(* PLC project emC-LUC-BS-Temp, PHOENIX CONTACT Software MULTIPROG 5.51 *)
(* stored: companyURL https://www.phoenixcontact-software.com, creationDateTime 2020-12-01T16:35:25, version 1606836925, modificationDateTime 2020-12-01T16:35:25 *)

TYPE TDC_DATA : ARRAY[0..199] OF BYTE;
END_TYPE

TYPE TDC : STRUCT
  transmit : BOOL;
  COT : USINT;
  confirm : BOOL;
  COTDesc : USINT;
  intOriginator : USINT;
  protocolType : USINT;
  totalNoOfSegments : USINT;
  currentSegment : USINT;
  lenOfData : UINT;
  data : TDC_DATA;
END_STRUCT;
END_TYPE

TYPE ThresholdType : (None, Integrated, Absolute) INT;
END_TYPE

TYPE COT : STRUCT
  Act : BOOL;
  ActCon : BOOL;
  Deact : BOOL;
  DeactCon : BOOL;
  ActTerm : BOOL;
END_STRUCT;
END_TYPE

TYPE Timestamp : STRUCT
  Milliseconds : UINT;
  Minutes : USINT;
  IV : BOOL;
  Hours : USINT;
  Summertime : BOOL;
  DayOfMonth : USINT;
  DayOfWeek : USINT;
  Month : USINT;
  Year : USINT;
END_STRUCT;
END_TYPE

TYPE AMI : STRUCT
  Value : INT;
  OV : BOOL;
  BL : BOOL;
  SB : BOOL;
  NT : BOOL;
  IV : BOOL;
  TR : BOOL;
  TimeTag : Timestamp;
  COT : USINT;
  FILL : BOOL;
END_STRUCT;
END_TYPE

TYPE ASO : STRUCT
  SE : BOOL;
  EX : BOOL;
  AQ : BOOL;
  QU : BYTE;
  Value : INT;
  COT : USINT;
  COTDesc : USINT;
  intOriginator : USINT;
END_STRUCT;
END_TYPE

TYPE BSI08 : STRUCT
  Value : BYTE;
  OV : BOOL;
  BL : BOOL;
  SB : BOOL;
  NT : BOOL;
  IV : BOOL;
  TimeTag : Timestamp;
  COT : USINT;
  FILL : BOOL;
END_STRUCT;
END_TYPE

TYPE BSI16 : STRUCT
  Value : WORD;
  OV : BOOL;
  BL : BOOL;
  SB : BOOL;
  NT : BOOL;
  IV : BOOL;
  FILL1 : BOOL;
  TimeTag : Timestamp;
  COT : USINT;
  FILL2 : BOOL;
END_STRUCT;
END_TYPE

TYPE BSI32 : STRUCT
  Value : DWORD;
  OV : BOOL;
  BL : BOOL;
  SB : BOOL;
  NT : BOOL;
  IV : BOOL;
  FILL1 : BOOL;
  TimeTag : Timestamp;
  COT : USINT;
  FILL2 : BOOL;
END_STRUCT;
END_TYPE

TYPE BSO01 : STRUCT
  SE : BOOL;
  EX : BOOL;
  AQ : BOOL;
  QU : BYTE;
  Value : BOOL;
  COT : USINT;
  COTDesc : USINT;
  intOriginator : USINT;
END_STRUCT;
END_TYPE

TYPE BSO02 : STRUCT
  SE : BOOL;
  EX : BOOL;
  AQ : BOOL;
  QU : BYTE;
  Value : BYTE;
  COT : USINT;
  COTDesc : USINT;
  intOriginator : USINT;
END_STRUCT;
END_TYPE

TYPE BSO08 : STRUCT
  SE : BOOL;
  EX : BOOL;
  AQ : BOOL;
  QU : BYTE;
  Value : BYTE;
  COT : USINT;
  COTDesc : USINT;
  intOriginator : USINT;
END_STRUCT;
END_TYPE

TYPE BSO16 : STRUCT
  SE : BOOL;
  EX : BOOL;
  AQ : BOOL;
  QU : BYTE;
  Value : WORD;
  COT : USINT;
  COTDesc : USINT;
  intOriginator : USINT;
END_STRUCT;
END_TYPE

TYPE DCO : STRUCT
  SE : BOOL;
  EX : BOOL;
  AQ : BOOL;
  QU : BYTE;
  Value : BYTE;
  COT : USINT;
  COTDesc : USINT;
  intOriginator : USINT;
END_STRUCT;
END_TYPE

TYPE DMI08 : STRUCT
  Value : WORD;
  OV : BOOL;
  BL : BOOL;
  SB : BOOL;
  NT : BOOL;
  IV : BOOL;
  FILL1 : BOOL;
  TimeTag : Timestamp;
  COT : USINT;
  FILL2 : BOOL;
END_STRUCT;
END_TYPE

TYPE DMI16 : STRUCT
  Value : WORD;
  OV : BOOL;
  BL : BOOL;
  SB : BOOL;
  NT : BOOL;
  IV : BOOL;
  FILL1 : BOOL;
  TimeTag : Timestamp;
  COT : USINT;
  FILL2 : BOOL;
END_STRUCT;
END_TYPE

TYPE DPI : STRUCT
  Value : BYTE;
  BL : BOOL;
  SB : BOOL;
  NT : BOOL;
  IV : BOOL;
  FILL1 : BOOL;
  TimeTag : Timestamp;
  COT : USINT;
  FILL2 : BOOL;
END_STRUCT;
END_TYPE

TYPE DSO08 : STRUCT
  SE : BOOL;
  EX : BOOL;
  AQ : BOOL;
  QU : BYTE;
  Value : INT;
  COT : USINT;
  COTDesc : USINT;
  intOriginator : USINT;
END_STRUCT;
END_TYPE

TYPE DSO16 : STRUCT
  SE : BOOL;
  EX : BOOL;
  AQ : BOOL;
  QU : BYTE;
  Value : INT;
  COT : USINT;
  COTDesc : USINT;
  intOriginator : USINT;
END_STRUCT;
END_TYPE

TYPE EPI : STRUCT
  Value : BYTE;
  EI : BOOL;
  BL : BOOL;
  SB : BOOL;
  NT : BOOL;
  IV : BOOL;
  SK1 : BOOL;
  SK2 : BOOL;
  SK3 : BOOL;
  SK4 : BOOL;
  SK5 : BOOL;
  SK6 : BOOL;
  SK7 : BOOL;
  SK8 : BOOL;
  ElpTime : UINT;
  FaultNo : UINT;
  TimeTag : Timestamp;
  COT : USINT;
  TypeVar : USINT;
  TR : BOOL;
  AQ : BOOL;
END_STRUCT;
END_TYPE

TYPE FSO : STRUCT
  SE : BOOL;
  EX : BOOL;
  AQ : BOOL;
  QU : BYTE;
  Value : REAL;
  COT : USINT;
  COTDesc : USINT;
  intOriginator : USINT;
END_STRUCT;
END_TYPE

TYPE ITI : STRUCT
  Value : DINT;
  SEQ : BYTE;
  CY : BOOL;
  CA : BOOL;
  IV : BOOL;
  TimeTag : Timestamp;
  COT : USINT;
  FILL : BOOL;
END_STRUCT;
END_TYPE

TYPE MFI : STRUCT
  Value : REAL;
  OV : BOOL;
  BL : BOOL;
  SB : BOOL;
  NT : BOOL;
  IV : BOOL;
  TR : BOOL;
  TimeTag : Timestamp;
  COT : USINT;
  FILL : BOOL;
END_STRUCT;
END_TYPE

TYPE RCO : STRUCT
  SE : BOOL;
  EX : BOOL;
  AQ : BOOL;
  QU : BYTE;
  Value : BYTE;
  COT : USINT;
  COTDesc : USINT;
  intOriginator : USINT;
END_STRUCT;
END_TYPE

TYPE SCO : STRUCT
  SE : BOOL;
  EX : BOOL;
  AQ : BOOL;
  QU : USINT;
  Value : BOOL;
  COT : USINT;
  COTDesc : USINT;
  intOriginator : USINT;
END_STRUCT;
END_TYPE

TYPE SEV : STRUCT
  Value : BOOL;
  IV : BOOL;
  TimeTag : Timestamp;
  COT : USINT;
  FILL2 : BOOL;
END_STRUCT;
END_TYPE

TYPE SPI : STRUCT
  Value : BOOL;
  BL : BOOL;
  SB : BOOL;
  NT : BOOL;
  IV : BOOL;
  FILL1 : BOOL;
  TimeTag : Timestamp;
  COT : USINT;
  FILL2 : BOOL;
END_STRUCT;
END_TYPE

TYPE SSC : STRUCT
  SE : BOOL;
  EX : BOOL;
  AQ : BOOL;
  QU : USINT;
  Value : BOOL;
  COT : USINT;
  COTDesc : USINT;
  intOriginator : USINT;
END_STRUCT;
END_TYPE

TYPE STI : STRUCT
  Value : USINT;
  Sign : BOOL;
  T : BOOL;
  OV : BOOL;
  BL : BOOL;
  NT : BOOL;
  SB : BOOL;
  IV : BOOL;
  TimeTag : Timestamp;
  COT : USINT;
  FILL : BOOL;
END_STRUCT;
END_TYPE

TYPE Structure_LUC_BESS_Pa : STRUCT
  PCtrlDeadbPa : REAL;
  PLimMaxPa : REAL;
  PLimMinPa : REAL;
  P_StoprampDownPa : REAL;
  P_StoprampUpPa : REAL;
  QCtrlDeadbPa : REAL;
  QLimMaxPa : REAL;
  QLimMinPa : REAL;
  Q_StoprampDownPa : REAL;
  Q_StoprampUpPa : REAL;
END_STRUCT;
END_TYPE

TYPE States : STRUCT
  sNotReady : INT;
  sReady : INT;
  sStarting : INT;
  sOnline : INT;
  sStopping : INT;
END_STRUCT;
END_TYPE

TYPE BattSMState : STRUCT
  StateNum : INT;
  BatInitializeSt : BOOL;
  BatNotReadySt : BOOL;
  BatReadySt : BOOL;
  BatStartingSt : BOOL;
  BatOnlineSt : BOOL;
  BatStoppingSt : BOOL;
END_STRUCT;
END_TYPE

TYPE BMSData : STRUCT
  Version : UINT;
  RacksNServiceCnt : USINT;
  TotalRackCnt : USINT;
  WatchDogError : BOOL;
  WatchDogCMD : UINT;
  WatchDogResp : UINT;
  HeartBeat : REAL;
  PartMinRackCnt : USINT;
  PartDiffVolt : REAL;
END_STRUCT;
END_TYPE

TYPE BMSSysConfig : STRUCT
  EStopProtEn : BOOL;
  EStopSPDEn : BOOL;
  FltResetCmdRejectEn : BOOL;
  DcSenFlEn : BOOL;
END_STRUCT;
END_TYPE

TYPE BMSMode : STRUCT
  ChargingSt : BOOL;
  DischargingSt : BOOL;
  BattRunningSt : BOOL;
  SwCloseRcvSt : BOOL;
  SwOpenRcvSt : BOOL;
  RkPartOnlineSt : BOOL;
  MdOfflineSt : BOOL;
  MdIdleSt : BOOL;
  MdReadySt : BOOL;
  EStopSPDSt : BOOL;
  EStopProtSt : BOOL;
  EStopPartSt : BOOL;
END_STRUCT;
END_TYPE

TYPE IntAlarm : STRUCT
  HealthySt : BOOL;
  FireSysOkSt : BOOL;
  CriticalAl : BOOL;
  NonCriticalAl : BOOL;
  WarningAl : BOOL;
  StateTOUT : BOOL;
  InitCommsFail : BOOL;
  MinRkCloseFail : BOOL;
  RkTripStart : BOOL;
  MinRkOnlineFail : BOOL;
  RkFailToOpen : BOOL;
  SysFireAl : BOOL;
  BmsLostCommsAl : BOOL;
  BankFault : BOOL;
  EStopAl : BOOL;
  ExtReadyStNotSetAl : BOOL;
  BattUSyncErrAl : BOOL;
  RkFail2Cls : BOOL;
  RkCntrFailAl : BOOL;
END_STRUCT;
END_TYPE

TYPE BMSAlarmSummary : STRUCT
  CriticalAl : BOOL;
  NonCriticalAl : BOOL;
  WarningAl : BOOL;
  RTUComAl : BOOL;
  RTUComFlt : BOOL;
  RkVoltImbAl : BOOL;
  SysStopAl : BOOL;
END_STRUCT;
END_TYPE

TYPE BMSAlarm : STRUCT
  ModuleUnderTempAl : BOOL;
  ModuleOverTempAl : BOOL;
  ModuleUnVoltAl : BOOL;
  ModuleOvVoltAl : BOOL;
  RackVoltRegAl : BOOL;
  RackTempRegAl : BOOL;
  AuxProtAl : BOOL;
  ChargeOperLimAl : BOOL;
  DischargeOperLimAl : BOOL;
  RackUnVoltAl : BOOL;
  RackOvVoltAl : BOOL;
  RackCommsAl : BOOL;
  TrayCommsAl : BOOL;
  DcCntrSensor1Al : BOOL;
  DcCntrSensor2Al : BOOL;
  FanFailAl : BOOL;
  ChargeOverCurrentAl : BOOL;
  DisChargeOverCurrentAl : BOOL;
  RackVSenseDiffAl : BOOL;
  RackFuseFailAl : BOOL;
  RackCurrentSenserFailAl : BOOL;
  RackPermanentUVAl : BOOL;
  DcCntr1Al : BOOL;
  DcCntr2Al : BOOL;
  DcSwCntFailAl : BOOL;
  CellVoltSenFailAl : BOOL;
  DCFuseSenserFailAl : BOOL;
END_STRUCT;
END_TYPE

TYPE BMSProt : STRUCT
  ModuleUnderTempAl : BOOL;
  ModuleOverTempAl : BOOL;
  ModuleUnVoltAl : BOOL;
  ModuleOvVoltAl : BOOL;
  RackVoltRegAl : BOOL;
  RackTempRegAl : BOOL;
  AuxProtAl : BOOL;
  ChargeOperLimAl : BOOL;
  DischargeOperLimAl : BOOL;
  RackUnVoltAl : BOOL;
  RackOvVoltAl : BOOL;
  RackCommsAl : BOOL;
  TrayCommsAl : BOOL;
  DcCntrSensor1Al : BOOL;
  DcCntrSensor2Al : BOOL;
  FanFailAl : BOOL;
  ChargeOverCurrentAl : BOOL;
  DisChargeOverCurrentAl : BOOL;
  RackVSenseDiffAl : BOOL;
  RackFuseFailAl : BOOL;
  RackCurrentSenserFailAl : BOOL;
  RackPermanentUVAl : BOOL;
  DcCntr1Al : BOOL;
  DcCntr2Al : BOOL;
  DcSwCntFailAl : BOOL;
  CellVoltSenFailAl : BOOL;
  DCFuseSenserFailAl : BOOL;
END_STRUCT;
END_TYPE

TYPE BMSSysMeasure : STRUCT
  UdcAct : REAL;
  IdcAct : REAL;
  BatPNomMaxAct : REAL;
  BatPNomMinAct : REAL;
  SocPctAct : REAL;
  SohAct : REAL;
  TempMaxAct : REAL;
  TempMinAct : REAL;
  ChrgMwhAct : REAL;
  DchrgMwhAct : REAL;
  CellMaxVolt : REAL;
  CellMinVolt : REAL;
  ServVolt : REAL;
  ServSoC : REAL;
END_STRUCT;
END_TYPE

TYPE BattSysMeasure : STRUCT
  UdcAct : REAL;
  IdcAct : REAL;
  NomPAct : REAL;
  NomEAct : REAL;
  BatPNomMaxAct : REAL;
  BatPNomMinAct : REAL;
  PAct : REAL;
  EAct : REAL;
  SocPctAct : REAL;
  SohAct : REAL;
  TempMaxAct : REAL;
  TempMinAct : REAL;
  SyncUSet : REAL;
END_STRUCT;
END_TYPE

TYPE Batt_Sys : STRUCT
  BattSMState : BattSMState;
  BMSSysConfig : BMSSysConfig;
  BMS_DATA : BMSData;
  BMS_Mode : BMSMode;
  BMSAlarmSummary : BMSAlarmSummary;
  BMSAlarm : BMSAlarm;
  BMSProt : BMSProt;
  Alarm : IntAlarm;
  BattSysMeasure : BattSysMeasure;
END_STRUCT;
END_TYPE

TYPE BMS_Sys : STRUCT
  BMS_DATA : BMSData;
  BMSSysConfig : BMSSysConfig;
  BMS_Mode : BMSMode;
  BMSAlarmSummary : BMSAlarmSummary;
  BMS_Alarm : BMSAlarm;
  BMS_Prot : BMSProt;
  BMS_Measure : BMSSysMeasure;
END_STRUCT;
END_TYPE

TYPE RkStatus : STRUCT
  RkOnlineSt : BOOL;
  RkOfflineSt : BOOL;
  RkInitSt : BOOL;
  Rk_Estop : BOOL;
  RkGridSwCmdRcv : BOOL;
END_STRUCT;
END_TYPE

TYPE RkData : STRUCT
  RkDcSw2On : BOOL;
  RkDcSw1On : BOOL;
  RkHeartBeat : INT;
  ModComFltPos : USINT;
  FanStatus : BOOL;
  Fuse1_On : BOOL;
  AuxProtect : BOOL;
END_STRUCT;
END_TYPE

TYPE RkAlarm : STRUCT
  RkCriticalAl : BOOL;
  RkNonCriticalAl : BOOL;
  RkWarningAl : BOOL;
  ModuleUT : BOOL;
  ModuleOT : BOOL;
  ModuleUV : BOOL;
  ModuleOV : BOOL;
  ModuleVImb : BOOL;
  Rk_ModuleComFail : BOOL;
  Rk_SystemComFail : BOOL;
  RkChargeOC : BOOL;
  RkDisChargeOC : BOOL;
  RkUV : BOOL;
  RkOV : BOOL;
  RkVSensDiff : BOOL;
  RkISensDiff : BOOL;
  RkFuseFail : BOOL;
  RkPermUV : BOOL;
  DcSw1SensFail : BOOL;
  DcSw2SensFail : BOOL;
  DcSw1Fail : BOOL;
  DcSw2Fail : BOOL;
  FanFail : BOOL;
  AuxProtFail : BOOL;
  CellChardeOpLim : BOOL;
  CellDisChargeOpLim : BOOL;
  ModulePcbUT : BOOL;
  ModulePcbOT : BOOL;
  DcSwCountFail : BOOL;
  CellVoltSenError : BOOL;
  DCContactSenFail : BOOL;
END_STRUCT;
END_TYPE

TYPE RkProtection : STRUCT
  ModuleUT : BOOL;
  ModuleOT : BOOL;
  ModuleUV : BOOL;
  ModuleOV : BOOL;
  ModuleVImb : BOOL;
  Rk_ModuleComFail : BOOL;
  Rk_SystemComFail : BOOL;
  RkChargeOC : BOOL;
  RkDisChargeOC : BOOL;
  RkUV : BOOL;
  RkOV : BOOL;
  RkVSensDiff : BOOL;
  RkISensDiff : BOOL;
  RkFuseFail : BOOL;
  RkPermUV : BOOL;
  DcSw1SensFail : BOOL;
  DcSw2SensFail : BOOL;
  DcSw1Fail : BOOL;
  DcSw2Fail : BOOL;
  FanFail : BOOL;
  AuxProtFail : BOOL;
  CellChardeOpLim : BOOL;
  CellDisChargeOpLim : BOOL;
  ModulePcbUT : BOOL;
  ModulePcbOT : BOOL;
  DcSwCountFail : BOOL;
  CellVoltSenError : BOOL;
  DCContactSenFail : BOOL;
END_STRUCT;
END_TYPE

TYPE RkMeasure : STRUCT
  UAct : REAL;
  IAct : REAL;
  SocAct : REAL;
  SohAct : REAL;
  CellMax1UdcAct : REAL;
  CellMax1UdcModID : USINT;
  CellMax1UdcCellID : USINT;
  CellMin1UdcAct : REAL;
  CellMin1UdcModID : REAL;
  CellMin1UdcCellID : REAL;
  CellMax2UdcAct : REAL;
  CellMax2UdcModID : USINT;
  CellMax2UdcCellID : REAL;
  CellMin2UdcAct : REAL;
  CellMin2UdcModID : REAL;
  CellMin2UdcCellID : REAL;
  CellMax1TempAct : REAL;
  CellMax1TempModID : USINT;
  CellMax1TempCellID : USINT;
  CellMin1TempAct : REAL;
  CellMin1TempModID : USINT;
  CellMin1TempCellID : USINT;
  CellMax2TempAct : REAL;
  CellMax2TempModID : USINT;
  CellMax2TempCellID : USINT;
  CellMin2TempAct : REAL;
  CellMin2TempModID : USINT;
  CellMin2TempCellID : USINT;
  CellAvgUdcAct : REAL;
  CellAvgTAct : REAL;
  ChrgLimSet : REAL;
  DchrgLimSet : REAL;
  IAvgAct : REAL;
END_STRUCT;
END_TYPE

TYPE Batt_RackStruct : STRUCT
  Data : RkData;
  Status : RkStatus;
  Alarm : RkAlarm;
  Protection : RkProtection;
  Measure : RkMeasure;
END_STRUCT;
END_TYPE

TYPE BMS_RackArray : ARRAY[1..32] OF Batt_RackStruct;
END_TYPE

TYPE Batt_Rack : STRUCT
  OnlineCnt : USINT;
  Ok2ClsCnt : USINT;
  Batt_Rack_Array : BMS_RackArray;
END_STRUCT;
END_TYPE

TYPE BkStatus : STRUCT
  BkHealthySt : BOOL;
END_STRUCT;
END_TYPE

TYPE BkAlarm : STRUCT
  CriticalAl : BOOL;
  NonCriticalAl : BOOL;
  WarningAl : BOOL;
  FireAl : BOOL;
  HvACAl : BOOL;
END_STRUCT;
END_TYPE

TYPE BkMeasures : STRUCT
  TotalRkCnt : USINT;
  RkOnlineCnt : USINT;
  AvgIdcAct : REAL;
  AvgSocAct : REAL;
  AvgSohAct : REAL;
  AvgTempAct : REAL;
  AvgUdcAct : REAL;
  MaxUAct : REAL;
  MinUAct : REAL;
END_STRUCT;
END_TYPE

TYPE Bank : STRUCT
  Status : BkStatus;
  Alarm : BkAlarm;
  Measures : BkMeasures;
END_STRUCT;
END_TYPE

TYPE Batt_Bank_Array : ARRAY[1..32] OF Bank;
END_TYPE

TYPE CtrlStruct : STRUCT
  RackAllCtrl : UINT;
  RackAllReset : UINT;
  WatchDogQuery : UINT;
END_STRUCT;
END_TYPE

TYPE MbCtrlStruct : STRUCT
  MB_Polling : INT;
  BmsLostCommsAl : BOOL;
  OneFullRead : BOOL;
  All_RkRead_Done : BOOL;
  BMS_Ctrl : CtrlStruct;
END_STRUCT;
END_TYPE

TYPE MbusPa : STRUCT
  MessageTimeDelayPa : TIME;
  MbCommTOutPa : TIME;
  NbOfRackPa : INT;
  WatchDogMode : INT;
END_STRUCT;
END_TYPE

TYPE DerateLookUpPa : ARRAY[1..6] OF REAL;
END_TYPE

TYPE MapOfRackStruct : ARRAY[1..32] OF INT;
END_TYPE

TYPE BattPLCParamStruct : STRUCT
  NbOfRackPa : INT;
  NbOfBankPa : INT;
  MinPctOfRkPa : REAL;
  MapOfRackPa : MapOfRackStruct;
  InvDcBusUMinPa : REAL;
  InvDcBusUMaxPa : REAL;
  InvPActMinPa : REAL;
  InvPActMaxPa : REAL;
  BattSysSyncUBiasPa : REAL;
  BATT_SYSSyncRangePa : REAL;
  RacksStartingTimeoutPa : TIME;
  RacksStoppingTimeoutPa : TIME;
  ClockSyncIntervalPa : TIME;
  ClockSyncEnPA : BOOL;
  WatchDogMode : INT;
  BattRackNomEActPa : REAL;
  BattRackNomPActPa : REAL;
  EnDerateWrtSocPa : BOOL;
  EnDerateWrtTempPa : BOOL;
  DrtChrgOnSocLookUpSocPa : DerateLookUpPa;
  DrtChrgOnSocLookUpDrtPa : DerateLookUpPa;
  DrtDChrgOnSocLookUpSocPa : DerateLookUpPa;
  DrtDChrgOnSocLookUpDrtPa : DerateLookUpPa;
  DerateTempLookUpTempPa : DerateLookUpPa;
  DerateTempLookUpDeratePa : DerateLookUpPa;
END_STRUCT;
END_TYPE

TYPE ModbusArray_Bat : ARRAY[0..199] OF WORD;
END_TYPE

TYPE RealArray_Bat : ARRAY[0..199] OF REAL;
END_TYPE

TYPE Array_of_MBusReadArray : ARRAY[0..31] OF ModbusArray_Bat;
END_TYPE

TYPE SchedAutomaticGeneratedDT_0001 : ARRAY[0..109] OF DINT;
END_TYPE

TYPE SchedAutomaticGeneratedDT_0002 : ARRAY[0..109] OF LREAL;
END_TYPE

TYPE SchedAutomaticGeneratedDT_0003 : ARRAY[0..99] OF LREAL;
END_TYPE

TYPE SchedAutomaticGeneratedDT_0004 : ARRAY[0..99] OF LREAL;
END_TYPE

TYPE SchedAutomaticGeneratedDT_0005 : ARRAY[0..9] OF SINT;
END_TYPE

TYPE SchedAutomaticGeneratedDT_0006 : ARRAY[0..9] OF BOOL;
END_TYPE

TYPE SchedAutomaticGeneratedDT_0007 : ARRAY[0..9] OF DINT;
END_TYPE

TYPE SchedAutomaticGeneratedDT_0008 : ARRAY[0..9] OF DINT;
END_TYPE

TYPE SchedAutomaticGeneratedDT_0009 : ARRAY[0..9] OF DINT;
END_TYPE

TYPE SchedAutomaticGeneratedDT_0010 : ARRAY[0..9] OF DINT;
END_TYPE

TYPE SchedAutomaticGeneratedDT_0011 : ARRAY[0..9] OF BOOL;
END_TYPE

TYPE SchedAutomaticGeneratedDT_0012 : ARRAY[0..9] OF BOOL;
END_TYPE

TYPE SchedAutomaticGeneratedDT_0013 : ARRAY[0..9] OF BOOL;
END_TYPE

TYPE SchedAutomaticGeneratedDT_0014 : ARRAY[0..9] OF REAL;
END_TYPE

TYPE SchedAutomaticGeneratedDT_0015 : ARRAY[0..9] OF DINT;
END_TYPE

TYPE SchedAutomaticGeneratedDT_0016 : ARRAY[0..15] OF BOOL;
END_TYPE

TYPE SchedAutomaticGeneratedDT_0017 : ARRAY[0..9] OF DINT;
END_TYPE

TYPE TIMER_Bat : STRUCT
  CountTick_t : DINT;
  Operate_t : BOOL;
  Started_t : BOOL;
  Expired_t : BOOL;
END_STRUCT;
END_TYPE

TYPE WordArray : ARRAY[0..7] OF WORD;
END_TYPE

TYPE WordArray4 : ARRAY[0..3] OF WORD;
END_TYPE

TYPE emCSMLog : ARRAY[0..50] OF STRING(80);
END_TYPE

TYPE ExtIntESM : STRUCT
  ManualMd : BOOL;
  OperatorMd : BOOL;
  AutoMd : BOOL;
  OnlineSt : BOOL;
  RunningSt : BOOL;
  HealthySt : BOOL;
  OpStartCmd : BOOL;
  OpStopCmd : BOOL;
  AutoStartCmd : BOOL;
  AutoStopCmd : BOOL;
  SchedulerStartStopCmd : BOOL;
  ResetCmd : BOOL;
  StopRampSt : BOOL;
  CriticalAlarm : BOOL;
  NonCriticalAlarm : BOOL;
  Warning : BOOL;
  AmILastGfm : BOOL;
  StartStopEnablePa : BOOL;
  SchedulerStartStopCmdEnPa : BOOL;
  StartingSt : BOOL;
  StoppingSt : BOOL;
  CoolingTimeActiveSt : BOOL;
  MinRunTimeActiveSt : BOOL;
  SchedulableSt : BOOL;
  FailedToStartAl : BOOL;
  FailedToStopAl : BOOL;
  GcStartCmdOut : BOOL;
  GcStopCmdOut : BOOL;
  GcStartStopCmdOut : BOOL;
  UnPSStartStopAlarm : BOOL;
  BatReadySt : BOOL;
  BatOnlineSt : BOOL;
  BatForceStop : BOOL;
  BatStartingSt : BOOL;
  BatStoppingSt : BOOL;
  BatEnCmdOut : BOOL;
  BatDisCmdOut : BOOL;
  BatEnDisCmdOut : BOOL;
  BatEmergencyStop : BOOL;
  OperatorStartCmdenabler : BOOL;
  OperatorStopCmdenabler : BOOL;
  AutoStartCmdenabler : BOOL;
  AutoStopCmdenabler : BOOL;
END_STRUCT;
END_TYPE

TYPE Pm : STRUCT
  FAct : REAL;
  UAct : REAL;
  PAct : REAL;
  QAct : REAL;
  Pf : REAL;
  I1 : REAL;
  I3 : REAL;
  I2 : REAL;
  U12 : REAL;
  U23 : REAL;
  U31 : REAL;
  F2Act : REAL;
  U2Act : REAL;
  SlipFreq : REAL;
  DeltaPhase : REAL;
  PmHealth : BOOL;
  PmLostComms : BOOL;
END_STRUCT;
END_TYPE

TYPE ModbusArrayPS : ARRAY[0..199] OF WORD;
END_TYPE

TYPE RealArrayPS : ARRAY[0..199] OF REAL;
END_TYPE

TYPE Query : STRUCT
  DisableSt : BOOL;
  Transmit : BOOL;
  StartReg : UINT;
  NumberReg : UINT;
  FunctionCode : INT;
  Cfg_ByteSwap : BOOL;
  Cfg_ConvType : INT;
  Cfg_TimeoutComm : TIME;
  Cfg_TimePoll : TIME;
  QueryIDNum : INT;
  Priority : INT;
  QType : INT;
  QuerySignalsDesc : STRING(80);
END_STRUCT;
END_TYPE

TYPE QueryArray : ARRAY[1..20] OF Query;
END_TYPE

TYPE FaultFlg : STRUCT
  Estp : BOOL;
  ACOverCurrent : BOOL;
  DCOverCurrent : BOOL;
  DCOverVoltage : BOOL;
  PDOverTemp : BOOL;
  InvOverTemp : BOOL;
  CmdMsg : BOOL;
  DCUnderVolt : BOOL;
  ACOverVolt : BOOL;
  IllegalTrans : BOOL;
  EEHeat : BOOL;
  EESction : BOOL;
  Cool : BOOL;
  TimedOverLoadAC : BOOL;
  TimedOverLoadDC : BOOL;
  ICOL : BOOL;
  CtlBdVolt : BOOL;
  PChImbal : BOOL;
  DiDt : BOOL;
  CoolingFlw : BOOL;
  ThrmOverLoad : BOOL;
  Fan : BOOL;
  POR : BOOL;
  Condensation : BOOL;
  I2C : BOOL;
  ExternalInhibit : BOOL;
  GroundFault : BOOL;
  Fuse : BOOL;
  Rsvd28 : BOOL;
  ACDisconnect : BOOL;
  Rsvd30 : BOOL;
  Rsvd31 : BOOL;
END_STRUCT;
END_TYPE

TYPE WrnFlgs : STRUCT
  CANW : BOOL;
  CANEP : BOOL;
  Thrm : BOOL;
  Fan : BOOL;
  EeSaveActive : BOOL;
  LocNetMismatch : BOOL;
  RemNetMismatch : BOOL;
  Condensation : BOOL;
  I2C : BOOL;
  ExternalInhibit : BOOL;
  MaintReqd : BOOL;
  GroundFault : BOOL;
  Fuse : BOOL;
  ACDisconnect : BOOL;
  Rsvd14 : BOOL;
  Rsvd15 : BOOL;
  Rsvd16 : BOOL;
  Rsvd17 : BOOL;
  Rsvd18 : BOOL;
  Rsvd19 : BOOL;
  Rsvd20 : BOOL;
  Rsvd21 : BOOL;
  Rsvd22 : BOOL;
  Rsvd23 : BOOL;
  Rsvd24 : BOOL;
  Rsvd25 : BOOL;
  Rsvd26 : BOOL;
  Rsvd27 : BOOL;
  Rsvd28 : BOOL;
  Rsvd29 : BOOL;
  Rsvd30 : BOOL;
  Rsvd31 : BOOL;
END_STRUCT;
END_TYPE

TYPE PS : STRUCT
  GCRunningSt : BOOL;
  GCHealthy : BOOL;
  GCStartingSt : BOOL;
  GCReadySt : BOOL;
  GCGridFollowing : BOOL;
  GCFaultSt : BOOL;
  GCGridForming : BOOL;
  GCAreaEPSLost : BOOL;
  GCChargingSt : BOOL;
  GCRideThru : BOOL;
  GCTransitionActiveSt : BOOL;
  GCGndFault : BOOL;
  GCDCOverU : BOOL;
  GCACDisconnect : BOOL;
  GCDCDisconnect : BOOL;
  GCDCGridDisconnect : BOOL;
  GCCabinetOpen : BOOL;
  GCManualShutdown : BOOL;
  GCOverTemp : BOOL;
  GCOverF : BOOL;
  GCUnderF : BOOL;
  GCACOverVolt : BOOL;
  GCACUnderVolt : BOOL;
  GCBlownFuse : BOOL;
  GCUnderTemp : BOOL;
  GCMemLoss : BOOL;
  GCHWTestFailed : BOOL;
  PSStateWord : INT;
  GCPAct : REAL;
  GCFAct : REAL;
  GCSNomAct : REAL;
  GCQAct : REAL;
  GCPF : REAL;
  GCEAct : REAL;
  TempAct : REAL;
  IGBTTempaAct : REAL;
  TrafoTempAct : REAL;
  OTTempAct : REAL;
  GCA : REAL;
  GCAPhA : REAL;
  GCAPhB : REAL;
  GCAPhC : REAL;
  GCUAct12 : REAL;
  GCUAct23 : REAL;
  GCUAct13 : REAL;
  GCUAct1N : REAL;
  GCUAct2N : REAL;
  GCUAct3N : REAL;
  GCUAct : REAL;
  GCABBCtrlWrongConfig : BOOL;
  GCABBCtrlReady : BOOL;
  GCABBCtrlStartingSt : BOOL;
  GCABBCtrlVGMActiveSt : BOOL;
  GCABBCtrlGSMActiveSt : BOOL;
  GCABBCtrlError : BOOL;
  GCABBCtrlStoppingSt : BOOL;
  GCABBCtrlIslanded : BOOL;
  ABBStateWord : INT;
  GCABBErrorID : REAL;
  GCLostComms : BOOL;
  GCCommsOk : BOOL;
  GCHardwareenablestatus : BOOL;
  GCACPowerAvailable : BOOL;
  GCDCPowerAvailable : BOOL;
  GCPowerCircuitEnabled : BOOL;
  GCMX1relaystatus : BOOL;
  GCMX2relaystatus : BOOL;
  GCPrechargestatus : BOOL;
  GCK2Relaystatus : BOOL;
  GCControlcommandsvalid : BOOL;
  GCPowercommandValid : BOOL;
  GCCurrentcommandValid : BOOL;
  GCPhaserotationstatus : BOOL;
  GCLinevoltagedetected : BOOL;
  GCUnused : BOOL;
  GCRemoteACPowerAvailable : BOOL;
  GCRemotephaserotationstatus : BOOL;
  GCRemoteLineVoltageDetected : BOOL;
  GCDI1Status : BOOL;
  GCDI2Status : BOOL;
  GCDI3Status : BOOL;
  GCDI4Status : BOOL;
  GCDO1Status : BOOL;
  GCDO2Status : BOOL;
  GCDO3Status : BOOL;
  GCDO4Status : BOOL;
  GCDClinkRefCmdValid : BOOL;
  GCPumpRunning : BOOL;
  GCPumpFault : BOOL;
  GCABBLostCommsStop : BOOL;
  CtrlSystemReady : BOOL;
  GCSysFltCode : UINT;
  GCFltFlgs : FaultFlg;
  GCWrnFlgs : WrnFlgs;
  CriticalAlarm : BOOL;
  NonCriticalAlarm : BOOL;
  Warning : BOOL;
  GCreconnectDelay : BOOL;
  GCMomentCessation : BOOL;
  GCInhibited : BOOL;
END_STRUCT;
END_TYPE

TYPE PS_Out_EXTINT : STRUCT
  QueryIn : Query;
  NumOfQueriesP2 : INT;
  QueryActPayload : TDC_DATA;
END_STRUCT;
END_TYPE

TYPE PS_In_EXTINT : STRUCT
  ActQueryOut : INT;
  PQueryExecOrder : WORD;
  WriteQStopped : BOOL;
  ConfigLogicReadOut : ModbusArrayPS;
  CmdBitsReadedchanged : BOOL;
END_STRUCT;
END_TYPE

TYPE FdxT : ARRAY[0..10] OF REAL;
END_TYPE

TYPE Column : ARRAY[1..4] OF REAL;
END_TYPE

TYPE Jacob : ARRAY[1..4] OF Column;
END_TYPE

TYPE Arr150BOOL : ARRAY[0..150] OF BOOL;
END_TYPE

TYPE Arr150REAL : ARRAY[0..150] OF REAL;
END_TYPE

TYPE GTG : STRUCT
  OnlineSt : BOOL;
  PAct : REAL;
  QAct : REAL;
  POvldAct : REAL;
  PMinAct : REAL;
  LsPMaxAct : REAL;
  PNomMinAct : REAL;
  PNomMaxAct : REAL;
  QNomMinAct : REAL;
  QNomMaxAct : REAL;
  ExtPSetActiveSt : BOOL;
  ExtQSetActiveSt : BOOL;
  HealthySt : BOOL;
  LostComms : BOOL;
  RunningSt : BOOL;
  FAct : REAL;
  UAct : REAL;
  LocalUACt : REAL;
END_STRUCT;
END_TYPE

TYPE GTGArray : ARRAY[0..5] OF GTG;
END_TYPE

TYPE PTG : STRUCT
  OnlineSt : BOOL;
  PAct : REAL;
  QAct : REAL;
  LocalOnlineSt : BOOL;
  ExtPActiveSt : BOOL;
  ExtQActiveSt : BOOL;
  LostComms : BOOL;
END_STRUCT;
END_TYPE

TYPE PTGArray : ARRAY[0..5] OF PTG;
END_TYPE

TYPE PSTG : STRUCT
  OnlineSt : BOOL;
  BatSocAct : REAL;
  PAct : REAL;
  QAct : REAL;
  SNomAct : REAL;
  LocalOnlineSt : BOOL;
  PNomMaxAct : REAL;
  PNomMinAct : REAL;
  ExtPActiveSt : BOOL;
  ExtQActiveSt : BOOL;
  Healthy : BOOL;
  LostComms : BOOL;
END_STRUCT;
END_TYPE

TYPE PSTGArray : ARRAY[0..5] OF PSTG;
END_TYPE

TYPE NTG : STRUCT
  NetQAct : REAL;
  NetPAct : REAL;
  NetUSet : REAL;
  NetFSet : REAL;
  NetPMaxSet : REAL;
  NetPMinSet : REAL;
  NetQMaxSet : REAL;
  NetQMinSet : REAL;
  SynchingSt : BOOL;
  ClosedSt : BOOL;
  OpenSt : BOOL;
  UAct : REAL;
  LostComms : BOOL;
END_STRUCT;
END_TYPE

TYPE NTGArray : ARRAY[0..5] OF NTG;
END_TYPE

TYPE FTG : STRUCT
  QAct : REAL;
  PAct : REAL;
  UAct : REAL;
  OnlineSt : BOOL;
END_STRUCT;
END_TYPE

TYPE FTGArray : ARRAY[0..10] OF FTG;
END_TYPE

TYPE GTPS : STRUCT
  OnlineSt : BOOL;
  PAct : REAL;
  QAct : REAL;
  POvldAct : REAL;
  PMinAct : REAL;
  LsPMaxAct : REAL;
  PNomMinAct : REAL;
  QNomMinAct : REAL;
  QNomMaxAct : REAL;
  GfmActiveSt : BOOL;
  GfwActiveSt : BOOL;
  ExtPSetActiveSt : BOOL;
  ExtQSetActiveSt : BOOL;
  HealthySt : BOOL;
  LostComms : BOOL;
END_STRUCT;
END_TYPE

TYPE GTPSArray : ARRAY[0..5] OF GTPS;
END_TYPE

TYPE PTPS : STRUCT
  OnlineSt : BOOL;
  PAct : REAL;
  QAct : REAL;
  ExtPActiveSt : BOOL;
  ExtQActiveSt : BOOL;
  LostComms : BOOL;
END_STRUCT;
END_TYPE

TYPE PTPSArray : ARRAY[0..5] OF PTPS;
END_TYPE

TYPE PSTPS : STRUCT
  OnlineSt : BOOL;
  StartingSt : BOOL;
  PAct : REAL;
  QAct : REAL;
  SNomAct : REAL;
  PsENomAct : REAL;
  PNomMaxAct : REAL;
  PNomMinAct : REAL;
  PLimMaxAct : REAL;
  PLimMinAct : REAL;
  QLimMaxAct : REAL;
  QLimMinAct : REAL;
  ExtPActiveSt : BOOL;
  ExtQActiveSt : BOOL;
  GfmActiveSt : BOOL;
  GfwActiveSt : BOOL;
  PsRestartActiveSt : BOOL;
  PmEAct : REAL;
  LostComms : BOOL;
END_STRUCT;
END_TYPE

TYPE PSTPSArray : ARRAY[0..5] OF PSTPS;
END_TYPE

TYPE NTPS : STRUCT
  NetQAct : REAL;
  NetUAct : REAL;
  NetPAct : REAL;
  NetUSet : REAL;
  NetFSet : REAL;
  NetPMaxSet : REAL;
  NetPMinSet : REAL;
  NetQMaxSet : REAL;
  NetQMinSet : REAL;
  SynchingSt : BOOL;
  OnlineSt : BOOL;
  NetUState : REAL;
  LostComms : BOOL;
END_STRUCT;
END_TYPE

TYPE NTPSArray : ARRAY[0..5] OF NTPS;
END_TYPE

TYPE FTPS : STRUCT
  QAct : REAL;
  PAct : REAL;
  UAct : REAL;
  OnlineSt : BOOL;
END_STRUCT;
END_TYPE

TYPE FTPSArray : ARRAY[0..10] OF FTPS;
END_TYPE

TYPE GTP : STRUCT
  OnlineSt : BOOL;
  PAct : REAL;
  QAct : REAL;
  PMinAct : REAL;
  GfmActiveSt : BOOL;
  ExtPSetActiveSt : BOOL;
  ExtQSetActiveSt : BOOL;
  LostComms : BOOL;
END_STRUCT;
END_TYPE

TYPE GTPArray : ARRAY[0..5] OF GTP;
END_TYPE

TYPE PTP : STRUCT
  OnlineSt : BOOL;
  PAct : REAL;
  QAct : REAL;
  PNomMaxAct : REAL;
  ExtPActiveSt : BOOL;
  ExtQActiveSt : BOOL;
  RePLimActiveSt : BOOL;
  PNomMinAct : REAL;
  LostComms : BOOL;
  RunningSt : BOOL;
  SNomAct : REAL;
  PkLopTestEnSt : BOOL;
  SmthActiveSt : BOOL;
  SmthTestEnSt : BOOL;
END_STRUCT;
END_TYPE

TYPE PTPArray : ARRAY[0..5] OF PTP;
END_TYPE

TYPE PSTP : STRUCT
  OnlineSt : BOOL;
  PAct : REAL;
  QAct : REAL;
  SNomAct : REAL;
  PsGfmOnlineSt : BOOL;
  PsENomAct : REAL;
  PNomMaxAct : REAL;
  PNomMinAct : REAL;
  PLimMinAct : REAL;
  ExtPActiveSt : BOOL;
  ExtQActiveSt : BOOL;
  GfmActiveSt : BOOL;
  PmEAct : REAL;
  LostComms : BOOL;
END_STRUCT;
END_TYPE

TYPE PSTPArray : ARRAY[0..5] OF PSTP;
END_TYPE

TYPE NTP : STRUCT
  OnlineSt : BOOL;
  NetQAct : REAL;
  NetPAct : REAL;
  NetPMaxSet : REAL;
  NetPMinSet : REAL;
  NetQMaxSet : REAL;
  NetQMinSet : REAL;
  ClosedSt : BOOL;
  OpenSt : BOOL;
  LostComms : BOOL;
END_STRUCT;
END_TYPE

TYPE NTPArray : ARRAY[0..5] OF NTP;
END_TYPE

TYPE FTP : STRUCT
  QAct : REAL;
  PAct : REAL;
  UAct : REAL;
  OnlineSt : BOOL;
END_STRUCT;
END_TYPE

TYPE FTPArray : ARRAY[0..10] OF FTP;
END_TYPE

TYPE GTN : STRUCT
  PNomAct : REAL;
  PNomPa : REAL;
  OnlineSt : BOOL;
  LostComms : BOOL;
END_STRUCT;
END_TYPE

TYPE GTNArray : ARRAY[0..5] OF GTN;
END_TYPE

TYPE PSTN : STRUCT
  PNomAct : REAL;
  PNomPa : REAL;
  OnlineSt : BOOL;
  LostComms : BOOL;
END_STRUCT;
END_TYPE

TYPE PSTNArray : ARRAY[0..5] OF PSTN;
END_TYPE

TYPE NTN : STRUCT
  PAct : REAL;
  QAct : REAL;
  DeltaU : REAL;
  DeltaF : REAL;
  Deltath : REAL;
  OpenSt : BOOL;
  CloseSt : BOOL;
  SyncFIncSt : BOOL;
  SyncFDecSt : BOOL;
  SyncUIncSt : BOOL;
  SyncUDecSt : BOOL;
  OnlineSt : BOOL;
  LostComms : BOOL;
END_STRUCT;
END_TYPE

TYPE NTNArray : ARRAY[0..5] OF NTN;
END_TYPE

TYPE FTN : STRUCT
  QAct : REAL;
  PAct : REAL;
  UAct : REAL;
  OnlineSt : BOOL;
END_STRUCT;
END_TYPE

TYPE FTNArray : ARRAY[0..10] OF FTN;
END_TYPE

TYPE Task_Name_Typ : ARRAY[0..9] OF BYTE;
END_TYPE

TYPE Extended_Task_Info : STRUCT
  TaskName : Task_Name_Typ;
  TaskPrio : INT;
  undocumented_0 : INT;
  TaskPeriod : INT;
  TaskStack : INT;
  unused_1 : INT;
  TaskWatchdog : INT;
  undocumented_2 : INT;
  undocumented_3 : INT;
  undocumented_4 : INT;
  CurDuration : INT;
  MinDuration : INT;
  MaxDuration : INT;
  undocumented_5 : INT;
  CurDelay : INT;
  MinDelay : INT;
  MaxDelay : INT;
END_STRUCT;
END_TYPE

TYPE ModbusArray : ARRAY[0..199] OF WORD;
END_TYPE

TYPE RealArray : ARRAY[0..199] OF REAL;
END_TYPE

TYPE MBSlaveWordData : ARRAY[0..3500] OF WORD;
END_TYPE

TYPE MBSlaveRealData : ARRAY[0..3500] OF REAL;
END_TYPE

TYPE BatSimSysData : ARRAY[0..39] OF WORD;
END_TYPE

TYPE BatSimRackData : ARRAY[0..59] OF WORD;
END_TYPE

TYPE RackDataArray : ARRAY[1..32] OF BatSimRackData;
END_TYPE

TYPE BatSimMBData : STRUCT
  Sys_Data : BatSimSysData;
  Rack_Data : RackDataArray;
END_STRUCT;
END_TYPE

TYPE BatSimBMSData : STRUCT
  Version : UINT;
  RacksNServiceCnt : USINT;
  TotalRackCnt : USINT;
  WatchDogResp : REAL;
  HeartBeat : REAL;
  PartMinRackCnt : USINT;
  PartDiffVolt : REAL;
  EStopProtEn : BOOL;
  EStopSPDEn : BOOL;
  FltResetCmdRejectEn : BOOL;
  DcSenFlEn : BOOL;
END_STRUCT;
END_TYPE

TYPE BatSimBMSMode : STRUCT
  ChargingSt : BOOL;
  DischargingSt : BOOL;
  BattRunningSt : BOOL;
  SwCloseRcvSt : BOOL;
  SwOpenRcvSt : BOOL;
  RkPartOnlineSt : BOOL;
  MdOfflineSt : BOOL;
  MdIdleSt : BOOL;
  MdReadySt : BOOL;
  EStopSPDSt : BOOL;
  EStopProtSt : BOOL;
  EStopPartSt : BOOL;
END_STRUCT;
END_TYPE

TYPE BatSimBMSAlarm : STRUCT
  ModuleUnderTempAl : BOOL;
  ModuleOverTempAl : BOOL;
  ModuleUnVoltAl : BOOL;
  ModuleOvVoltAl : BOOL;
  RackVoltRegAl : BOOL;
  RackTempRegAl : BOOL;
  AuxProtAl : BOOL;
  ChargeOperLimAl : BOOL;
  DischargeOperLimAl : BOOL;
  RackUnVoltAl : BOOL;
  RackOvVoltAl : BOOL;
  RackCommsAl : BOOL;
  TrayCommsAl : BOOL;
  DcCntrSensor1Al : BOOL;
  DcCntrSensor2Al : BOOL;
  FanFailAl : BOOL;
  ChargeOverCurrentAl : BOOL;
  DisChargeOverCurrentAl : BOOL;
  RackVSenseDiffAl : BOOL;
  RackFuseFailAl : BOOL;
  RackCurrentSenserFailAl : BOOL;
  RackPermanentUVAl : BOOL;
  DcCntr1Al : BOOL;
  DcCntr2Al : BOOL;
  DcSwCntFailAl : BOOL;
  CellVoltSenFailAl : BOOL;
  DCFuseSenserFailAl : BOOL;
  RTUComAl : BOOL;
  RTUComFlt : BOOL;
  RkVoltImbAl : BOOL;
  SysStopAl : BOOL;
END_STRUCT;
END_TYPE

TYPE BatSimBMSProt : STRUCT
  ModuleUnderTempAl : BOOL;
  ModuleOverTempAl : BOOL;
  ModuleUnVoltAl : BOOL;
  ModuleOvVoltAl : BOOL;
  RackVoltRegAl : BOOL;
  RackTempRegAl : BOOL;
  AuxProtAl : BOOL;
  ChargeOperLimAl : BOOL;
  DischargeOperLimAl : BOOL;
  RackUnVoltAl : BOOL;
  RackOvVoltAl : BOOL;
  RackCommsAl : BOOL;
  TrayCommsAl : BOOL;
  DcCntrSensor1Al : BOOL;
  DcCntrSensor2Al : BOOL;
  FanFailAl : BOOL;
  ChargeOverCurrentAl : BOOL;
  DisChargeOverCurrentAl : BOOL;
  RackVSenseDiffAl : BOOL;
  RackFuseFailAl : BOOL;
  RackCurrentSenserFailAl : BOOL;
  RackPermanentUVAl : BOOL;
  DcCntr1Al : BOOL;
  DcCntr2Al : BOOL;
  DcSwCntFailAl : BOOL;
  CellVoltSenFailAl : BOOL;
  DCFuseSenserFailAl : BOOL;
END_STRUCT;
END_TYPE

TYPE BatSimSysMeasure : STRUCT
  UdcAct : REAL;
  IdcAct : REAL;
  SocPctAct : REAL;
  SohAct : REAL;
  TempMaxAct : REAL;
  TempMinAct : REAL;
  HumidtyAct : REAL;
  ChrgMwhAct : REAL;
  DchrgMwhAct : REAL;
  CellMaxVolt : REAL;
  CellMinVolt : REAL;
  ServVolt : REAL;
  ServSoC : REAL;
END_STRUCT;
END_TYPE

TYPE BatSimBMS_Sys : STRUCT
  BMS_DATA : BatSimBMSData;
  BMS_Mode : BatSimBMSMode;
  BMSP_Alarm : BatSimBMSAlarm;
  BMS_Prot : BatSimBMSProt;
  BMS_Measure : BatSimSysMeasure;
END_STRUCT;
END_TYPE

TYPE BatSimRkStatus : STRUCT
  RkOnlineSt : BOOL;
  RkOfflineSt : BOOL;
  RkInitSt : BOOL;
  Rk_Estop : BOOL;
  RkGridSwCmdRcv : BOOL;
END_STRUCT;
END_TYPE

TYPE BatSimRkData : STRUCT
  RkDcSw2On : BOOL;
  RkDcSw1On : BOOL;
  RkHeartBeat : INT;
  ModComFltPos : USINT;
  FanStatus : BOOL;
  Fuse1_On : BOOL;
  AuxProtect : BOOL;
END_STRUCT;
END_TYPE

TYPE BatSimRkAlarm : STRUCT
  ModuleUT : BOOL;
  ModuleOT : BOOL;
  ModuleUV : BOOL;
  ModuleOV : BOOL;
  ModuleVImb : BOOL;
  Rk_ModuleComFail : BOOL;
  Rk_SystemComFail : BOOL;
  RkChargeOC : BOOL;
  RkDisChargeOC : BOOL;
  RkUV : BOOL;
  RkOV : BOOL;
  RkVSensDiff : BOOL;
  RkISensDiff : BOOL;
  RkFuseFail : BOOL;
  RkPermUV : BOOL;
  DcSw1SensFail : BOOL;
  DcSw2SensFail : BOOL;
  DcSw1Fail : BOOL;
  DcSw2Fail : BOOL;
  FanFail : BOOL;
  AuxProtFail : BOOL;
  CellChardeOpLim : BOOL;
  CellDisChargeOpLim : BOOL;
  ModulePcbUT : BOOL;
  ModulePcbOT : BOOL;
  DcSwCountFail : BOOL;
  CellVoltSenError : BOOL;
  DCContactSenFail : BOOL;
END_STRUCT;
END_TYPE

TYPE BatSimRkProtection : STRUCT
  ModuleUT : BOOL;
  ModuleOT : BOOL;
  ModuleUV : BOOL;
  ModuleOV : BOOL;
  ModuleVImb : BOOL;
  Rk_ModuleComFail : BOOL;
  Rk_SystemComFail : BOOL;
  RkChargeOC : BOOL;
  RkDisChargeOC : BOOL;
  RkUV : BOOL;
  RkOV : BOOL;
  RkVSensDiff : BOOL;
  RkISensDiff : BOOL;
  RkFuseFail : BOOL;
  RkPermUV : BOOL;
  DcSw1SensFail : BOOL;
  DcSw2SensFail : BOOL;
  DcSw1Fail : BOOL;
  DcSw2Fail : BOOL;
  FanFail : BOOL;
  AuxProtFail : BOOL;
  CellChardeOpLim : BOOL;
  CellDisChargeOpLim : BOOL;
  ModulePcbUT : BOOL;
  ModulePcbOT : BOOL;
  DcSwCountFail : BOOL;
  CellVoltSenError : BOOL;
  DCContactSenFail : BOOL;
END_STRUCT;
END_TYPE

TYPE BatSimRkMeasure : STRUCT
  UAct : REAL;
  IAct : REAL;
  SocAct : REAL;
  SohAct : REAL;
  CellMax1UdcAct : REAL;
  CellMax1UdcModID : USINT;
  CellMax1UdcCellID : USINT;
  CellMin1UdcAct : REAL;
  CellMin1UdcModID : REAL;
  CellMin1UdcCellID : REAL;
  CellMax2UdcAct : REAL;
  CellMax2UdcModID : USINT;
  CellMax2UdcCellID : REAL;
  CellMin2UdcAct : REAL;
  CellMin2UdcModID : REAL;
  CellMin2UdcCellID : REAL;
  CellMax1TempAct : REAL;
  CellMax1TempModID : USINT;
  CellMax1TempCellID : USINT;
  CellMin1TempAct : REAL;
  CellMin1TempModID : USINT;
  CellMin1TempCellID : USINT;
  CellMax2TempAct : REAL;
  CellMax2TempModID : USINT;
  CellMax2TempCellID : USINT;
  CellMin2TempAct : REAL;
  CellMin2TempModID : USINT;
  CellMin2TempCellID : USINT;
  CellAvgUdcAct : REAL;
  CellAvgTAct : REAL;
  ChrgLimSet : REAL;
  DchrgLimSet : REAL;
  IAvgAct : REAL;
END_STRUCT;
END_TYPE

TYPE BatSimRackStruct : STRUCT
  Status : BatSimRkStatus;
  Data : BatSimRkData;
  Alarm : BatSimRkAlarm;
  Protection : BatSimRkProtection;
  Measure : BatSimRkMeasure;
END_STRUCT;
END_TYPE

TYPE BatSim_Rack_Array : ARRAY[1..32] OF BatSimRackStruct;
END_TYPE

TYPE LoadProfile : ARRAY[1..100] OF REAL;
END_TYPE

TYPE Fed_ModBus_In : STRUCT
  CloseCmd : BOOL;
  OpenCmd : BOOL;
  AlarmReset : BOOL;
END_STRUCT;
END_TYPE

TYPE Feeder_Var_IN : STRUCT
  uAct_Sys : REAL;
  GenLoading : REAL;
  GenCritAlarm : BOOL;
  FedPSet : REAL;
  FedQSet : REAL;
  FedCloseCmd : BOOL;
  FedOpenCmd : BOOL;
  FedResetCmd : BOOL;
END_STRUCT;
END_TYPE

TYPE Feeder_Param : STRUCT
  NbOfFedPa : INT;
  PScalarPa : REAL;
  QScalarPa : REAL;
  ScenarioSelectedPa : REAL;
  timelowPa : TIME;
  timehighPa : TIME;
END_STRUCT;
END_TYPE

TYPE Feeder_Out : STRUCT
  PAct : REAL;
  QAct : REAL;
  SAct : REAL;
  PfAct : REAL;
  U12Act : REAL;
  U23Act : REAL;
  U31Act : REAL;
  I1Act : REAL;
  I2Act : REAL;
  I3Act : REAL;
  Stat : BOOL;
  NCAlarm : BOOL;
  CritAlarm : BOOL;
  TRIP : BOOL;
  Eact : UDINT;
  EExportAct : UDINT;
  EImportAct : UDINT;
  KvarhAct : UDINT;
  ExportedKvarhAct : UDINT;
  ImportedKvarhAct : UDINT;
  U1nAct : REAL;
  U2nAct : REAL;
  U3nAct : REAL;
  U123AvgAct : REAL;
  WarningAl : BOOL;
  PermitToCloseSt : BOOL;
  CbTripSt : BOOL;
  IAvgAct : REAL;
  HealthySt : BOOL;
  UAct : REAL;
  ManualSt : BOOL;
END_STRUCT;
END_TYPE

TYPE Feeder_Struct : STRUCT
  Feeder_Param : Feeder_Param;
  Feeder_In : Feeder_Var_IN;
  Fed_ModBus_In : Fed_ModBus_In;
  Feeder_Out : Feeder_Out;
END_STRUCT;
END_TYPE

TYPE Feeder_Data : ARRAY[1..2] OF Feeder_Struct;
END_TYPE

TYPE Feeder_Summary : STRUCT
  PAct : REAL;
  QAct : REAL;
  OnlineSt : BOOL;
END_STRUCT;
END_TYPE

TYPE Grid_In : STRUCT
  CloseCmd : BOOL;
  OpenCmd : BOOL;
  AlarmReset : BOOL;
  CloseCmdSimGrid : BOOL;
  OpenCmdSimGrid : BOOL;
END_STRUCT;
END_TYPE

TYPE Grid_HMI_In : STRUCT
  CloseCmd : BOOL;
  OpenCmd : BOOL;
  AlarmReset : BOOL;
END_STRUCT;
END_TYPE

TYPE Grid_Param : STRUCT
  EInertia_GenPa : REAL;
  EInertiaPa : REAL;
  Sk_IslandPa : REAL;
  Sk_GridPa : REAL;
  FNomPa : REAL;
  UNomPa : REAL;
END_STRUCT;
END_TYPE

TYPE Grid_Out : STRUCT
  fAct : REAL;
  fAct_pu : REAL;
  uAct : REAL;
  uAct_pu : REAL;
  Stat : BOOL;
  CbTripSt : BOOL;
  PermitToCloseSt : BOOL;
  On : BOOL;
  TRIP : BOOL;
  Phase : REAL;
  PAct : REAL;
  QAct : REAL;
  SAct : REAL;
  PfAct : REAL;
  U12_util : REAL;
  U23_util : REAL;
  U31_util : REAL;
  U12Act : REAL;
  U23Act : REAL;
  U31Act : REAL;
  I1Act : REAL;
  I2Act : REAL;
  I3Act : REAL;
  Sync_stat : BOOL;
  CritAlarm : BOOL;
  NCAlarm : BOOL;
  WarningAl : BOOL;
  U123AvgAct : REAL;
  IAvgAct : REAL;
  EAct : UDINT;
  EExportAct : UDINT;
  EImportAct : UDINT;
  U1nAct : REAL;
  U2nAct : REAL;
  U3nAct : REAL;
  ExportKvarhAct : UDINT;
  ImportKvarhAct : UDINT;
  KvarhAct : UDINT;
  SyncCheckSt : BOOL;
  ManualSt : BOOL;
  HealthySt : BOOL;
END_STRUCT;
END_TYPE

TYPE Grid_HMI_Out : STRUCT
  BreakerClosedSt : BOOL;
  PAct : REAL;
  QAct : REAL;
  FAct : REAL;
  UAct : REAL;
  CritAlarm : BOOL;
  NCAlarm : BOOL;
END_STRUCT;
END_TYPE

TYPE Grid : STRUCT
  Grid_In : Grid_In;
  Grid_Param : Grid_Param;
  Grid_Out : Grid_Out;
  Grid_HMI_In : Grid_HMI_In;
  Grid_HMI_Out : Grid_HMI_Out;
END_STRUCT;
END_TYPE

TYPE Grid_Dat : ARRAY[1..2] OF Grid;
END_TYPE

TYPE Sys_Parameters : STRUCT
  FNomPa : REAL;
  UNomPa : REAL;
END_STRUCT;
END_TYPE

TYPE Sys_Data : STRUCT
  FAct : REAL;
  UAct : REAL;
  fAct_pu : REAL;
  uAct_pu : REAL;
  Grid_Stat : BOOL;
END_STRUCT;
END_TYPE

TYPE BMS_To_Gc : STRUCT
  BattOnlineSt : BOOL;
END_STRUCT;
END_TYPE

TYPE Gc_To_BMS : STRUCT
  PAct : REAL;
END_STRUCT;
END_TYPE

TYPE Gc_Param_In : STRUCT
  PQ_FU_RefSelPa : INT;
  FNomPa : REAL;
  UNomPa : REAL;
  SNomPa : REAL;
  fDroopPa : REAL;
  UDroopPa : REAL;
  TMotorPa : TIME;
  TExciterPa : TIME;
  P_UpPa : REAL;
  P_DownPa : REAL;
  PLimMinPa : REAL;
  PLimMaxPa : REAL;
  PinitPa : REAL;
  PNomPa : REAL;
  QLimMinPa : REAL;
  QLimMaxPa : REAL;
  QinitPa : REAL;
  QNomPa : REAL;
  OvPFactorPa : REAL;
  OvPLockInTPa : TIME;
  OvQFactorPa : REAL;
  OvQLockInTPa : TIME;
  OvUFactorPa : REAL;
  OvULockInTPa : TIME;
  OvFFactorPa : REAL;
  OvFLockInTPa : TIME;
  BrekarStatusInit : BOOL;
END_STRUCT;
END_TYPE

TYPE Gc_LuC_In : STRUCT
  StartCmd : BOOL;
  StopCmd : BOOL;
  AlarmReset : BOOL;
  FSet : REAL;
  USet : REAL;
  PSet : REAL;
  Qset : REAL;
  BreakerCloseCmd : BOOL;
  BreakerOpenCmd : BOOL;
  GridForming : BOOL;
  GrdFmg_Fctrl : BOOL;
  GrdFmg_Vctrl : BOOL;
  GrdFmg_Pctrl : BOOL;
  GrdFmg_Qctrl : BOOL;
  GrdFlw_Fsup : BOOL;
  GrdFlw_Vsup : BOOL;
  GrdFlw_Pctrl : BOOL;
  GrdFlw_Qctrl : BOOL;
  PLimMaxPa : REAL;
  PLimMinPa : REAL;
  QLimMaxPa : REAL;
  QLimMinPa : REAL;
  Enable : BOOL;
  FaultReset : BOOL;
  AllowGFWEnPa : BOOL;
  AllowGFMEnPa : BOOL;
END_STRUCT;
END_TYPE

TYPE Gc_HMI_In : STRUCT
  StartCmd : BOOL;
  StopCmd : BOOL;
  BreakerCloseCmd : BOOL;
  BreakerOpenCmd : BOOL;
  AlarmReset : BOOL;
  Sim_CritAl : BOOL;
  Sim_NonCritAl : BOOL;
  Sim_WarnAl : BOOL;
  EStop : BOOL;
END_STRUCT;
END_TYPE

TYPE Gc_LuC_Out : STRUCT
  PAct : REAL;
  QAct : REAL;
  SAct : REAL;
  OnLineSt : BOOL;
  RunningSt : BOOL;
  BreakerSt : BOOL;
  GCRunningSt : BOOL;
  GCHealthy : BOOL;
  GCStartingSt : BOOL;
  GCReadySt : BOOL;
  GCGridFollowing : BOOL;
  GCFaultSt : BOOL;
  GCGridForming : BOOL;
  GCAreaEPSLost : BOOL;
  GCChargingSt : BOOL;
  GCRideThru : BOOL;
  GCTransitionActiveSt : BOOL;
  GCGndFault : BOOL;
  GCDCOverU : BOOL;
  GCACDisconnect : BOOL;
  GCDCDisconnect : BOOL;
  GCDCGridDisconnect : BOOL;
  GCCabinetOpen : BOOL;
  GCManualShutdown : BOOL;
  GCOverTemp : BOOL;
  GCOverF : BOOL;
  GCUnderF : BOOL;
  GCACOverVolt : BOOL;
  GCACUnderVolt : BOOL;
  GCBlownFuse : BOOL;
  GCUnderTemp : BOOL;
  GCMemLoss : BOOL;
  GCHWTestFailed : BOOL;
  PSStateWord : INT;
  GCPAct : REAL;
  GCFAct : REAL;
  GCSNomAct : REAL;
  GCQAct : REAL;
  GCPF : REAL;
  GCEAct : REAL;
  TempAct : REAL;
  IGBTTempaAct : REAL;
  TrafoTempAct : REAL;
  OTTempAct : REAL;
  GCA : REAL;
  GCAPhA : REAL;
  GCAPhB : REAL;
  GCAPhC : REAL;
  GCUAct12 : REAL;
  GCUAct23 : REAL;
  GCUAct13 : REAL;
  GCUAct1N : REAL;
  GCUAct2N : REAL;
  GCUAct3N : REAL;
  GCUAct : REAL;
  GCABBCtrlWrongConfig : BOOL;
  GCABBCtrlReady : BOOL;
  GCABBCtrlStartingSt : BOOL;
  GCABBCtrlVGMActiveSt : BOOL;
  GCABBCtrlGSMActiveSt : BOOL;
  GCABBCtrlError : BOOL;
  GCABBCtrlStoppingSt : BOOL;
  GCABBCtrlIslanded : BOOL;
  ABBStateWord : INT;
  GCABBErrorID : REAL;
  GCLostComms : BOOL;
  GCCommsOk : BOOL;
  GCHardwareenablestatus : BOOL;
  GCACPowerAvailable : BOOL;
  GCDCPowerAvailable : BOOL;
  GCPowerCircuitEnabled : BOOL;
  GCMX1relaystatus : BOOL;
  GCMX2relaystatus : BOOL;
  GCPrechargestatus : BOOL;
  GCK2Relaystatus : BOOL;
  GCControlcommandsvalid : BOOL;
  GCPowercommandValid : BOOL;
  GCCurrentcommandValid : BOOL;
  GCPhaserotationstatus : BOOL;
  GCLinevoltagedetected : BOOL;
  GCUnused : BOOL;
  GCRemoteACPowerAvailable : BOOL;
  GCRemotephaserotationstatus : BOOL;
  GCRemoteLineVoltageDetected : BOOL;
  GCDI1Status : BOOL;
  GCDI2Status : BOOL;
  GCDI3Status : BOOL;
  GCDI4Status : BOOL;
  GCDO1Status : BOOL;
  GCDO2Status : BOOL;
  GCDO3Status : BOOL;
  GCDO4Status : BOOL;
  GCDClinkRefCmdValid : BOOL;
  GCPumpRunning : BOOL;
  GCPumpFault : BOOL;
  GCABBLostCommsStop : BOOL;
  CtrlSystemReady : BOOL;
  GCSysFltCode : UINT;
  GCFltFlgs : INT;
  GCWrnFlgs : INT;
  CriticalAlarm : BOOL;
  NonCriticalAlarm : BOOL;
  Warning : BOOL;
  GCreconnectDelay : BOOL;
  GCMomentCessation : BOOL;
  GCInhibited : BOOL;
END_STRUCT;
END_TYPE

TYPE Gc_HMI_Out : STRUCT
  PAct : REAL;
  QAct : REAL;
  UAct : REAL;
  FAct : REAL;
  IAvgAct : REAL;
  BreakerSt : BOOL;
  OnlineSt : BOOL;
END_STRUCT;
END_TYPE

TYPE Gc_Sys_Out : STRUCT
  FAct : REAL;
  UAct : REAL;
END_STRUCT;
END_TYPE

TYPE Gc_In : STRUCT
  Param : Gc_Param_In;
  LuC : Gc_LuC_In;
  BMS : BMS_To_Gc;
  HMI : Gc_HMI_In;
END_STRUCT;
END_TYPE

TYPE Gc_Out : STRUCT
  LuC : Gc_LuC_Out;
  BMS : Gc_To_BMS;
  HMI : Gc_HMI_Out;
  Sys : Gc_Sys_Out;
END_STRUCT;
END_TYPE

TYPE Gc_Struct : STRUCT
  In : Gc_In;
  Out : Gc_Out;
END_STRUCT;
END_TYPE

TYPE BatSimRkSM_In : STRUCT
  InService : BOOL;
  CloseCmd : BOOL;
  OpenCmd : BOOL;
  Alarm : BOOL;
END_STRUCT;
END_TYPE

TYPE BatSimRkSM_Out : STRUCT
  OnlineSt : BOOL;
  OfflineSt : BOOL;
  GridSwCmdRcv : BOOL;
END_STRUCT;
END_TYPE

TYPE BatSim_RkSMStruct : STRUCT
  In : BatSimRkSM_In;
  Out : BatSimRkSM_Out;
END_STRUCT;
END_TYPE

TYPE BatSim_RkSM : ARRAY[1..32] OF BatSim_RkSMStruct;
END_TYPE

TYPE BatSim_RkSM_IN : ARRAY[1..32] OF BatSimRkSM_In;
END_TYPE

TYPE BatSim_RkSM_Out : ARRAY[1..32] OF BatSimRkSM_Out;
END_TYPE

TYPE DerateLookUp : ARRAY[1..6] OF REAL;
END_TYPE

TYPE BMS_Param_In : STRUCT
  BatUNomPa : REAL;
  BatSNomPa : REAL;
  EInitPa : REAL;
  ENomPa : REAL;
  EnDerateWrtSocPa : BOOL;
  EnDerateWrtTempPa : BOOL;
  DrtChrgOnSocLookUpSocPa : DerateLookUp;
  DrtChrgOnSocLookUpDrtPa : DerateLookUp;
  DrtDChrgOnSocLookUpSocPa : DerateLookUp;
  DrtDChrgOnSocLookUpDrtPa : DerateLookUp;
  DerateTempLookUpTempPa : DerateLookUp;
  DerateTempLookUpDeratePa : DerateLookUp;
  BatPNomMinPa : REAL;
  BatPNomMaxPa : REAL;
  UMaxPa : REAL;
  UMinPa : REAL;
  TotalRackCntPa : USINT;
  PartMinRackCntPa : USINT;
END_STRUCT;
END_TYPE

TYPE BMS_LuC_In : STRUCT
  StartCmd : BOOL;
  StopCmd : BOOL;
  AlarmReset : BOOL;
  WatchDogQuery : REAL;
END_STRUCT;
END_TYPE

TYPE BMS_HMI_In : STRUCT
  StartCmd : BOOL;
  StopCmd : BOOL;
  AlarmReset : BOOL;
  Sim_CritAl : BOOL;
  Sim_NonCritAl : BOOL;
  Sim_WarnAl : BOOL;
  EStop : BOOL;
  TempMinAct : REAL;
  TempMaxAct : REAL;
  Sim_FireAl : BOOL;
  Rk_IN : BatSim_RkSM_IN;
END_STRUCT;
END_TYPE

TYPE BMS_Param_Out : STRUCT
  PQ_FU_RefSelPa : INT;
END_STRUCT;
END_TYPE

TYPE BMS_LuC_Out : STRUCT
  BatSim_Rack_Array : BatSim_Rack_Array;
  BatSimBMS_Sys : BatSimBMS_Sys;
END_STRUCT;
END_TYPE

TYPE BMS_HMI_Out : STRUCT
  PAct : REAL;
  QAct : REAL;
  UAct : REAL;
  IAct : REAL;
  OnlineSt : BOOL;
  OfflineSt : BOOL;
  Rk_Out : BatSim_RkSM_Out;
END_STRUCT;
END_TYPE

TYPE BMS_In : STRUCT
  Param : BMS_Param_In;
  LuC : BMS_LuC_In;
  Gc : Gc_To_BMS;
  HMI : BMS_HMI_In;
END_STRUCT;
END_TYPE

TYPE BMS_Out : STRUCT
  Param : BMS_Param_Out;
  LuC : BMS_LuC_Out;
  Gc : BMS_To_Gc;
  HMI : BMS_HMI_Out;
END_STRUCT;
END_TYPE

TYPE BMS_Struct : STRUCT
  In : BMS_In;
  Out : BMS_Out;
END_STRUCT;
END_TYPE

TYPE LineUP : STRUCT
  Gc : Gc_Struct;
  BMS : BMS_Struct;
END_STRUCT;
END_TYPE

TYPE Ps_LineUP : ARRAY[1..32] OF LineUP;
END_TYPE

TYPE Ps_Sum : STRUCT
  PsPAct : REAL;
  PsQAct : REAL;
  PsSAct : REAL;
  PsOnlineSt : BOOL;
  PsOfflineSt : BOOL;
  PsOnlineCnt : INT;
  PsOfflineCnt : INT;
END_STRUCT;
END_TYPE

TYPE DataQuery : ARRAY[0..30] OF WORD;
END_TYPE

TYPE QuerySim : STRUCT
  DisableSt : BOOL;
  Transmit : BOOL;
  StartReg : UINT;
  NumberReg : UINT;
  FunctionCode : INT;
  Cfg_ByteSwap : BOOL;
  Cfg_ConvType : INT;
  Cfg_TimeoutComm : TIME;
  Cfg_TimePoll : TIME;
  QueryIDNum : INT;
  Priority : INT;
  QType : INT;
  QuerySignalsDesc : STRING(80);
  Data : DataQuery;
END_STRUCT;
END_TYPE

TYPE QueryArraySim : ARRAY[1..20] OF QuerySim;
END_TYPE

TYPE MBSlaveBoolData : ARRAY[0..99] OF BOOL;
END_TYPE

TYPE Synch_Parameters : STRUCT
  NatGridUPa : REAL;
  NatGridfPa : REAL;
  GridNomUPa : REAL;
  NatGridNUPa : REAL;
  GridNomFPa : REAL;
  NatGridNomFPa : REAL;
  SlipfPa : REAL;
  MaxDiffUPa : REAL;
  TParallelTimePa : TIME;
  SynchModefPa : INT;
  SynchModeUPa : INT;
  FreqAdjChaPa : REAL;
  FMZeroTimePa : TIME;
  FMMinDTimePa : TIME;
  VAdjChaPa : REAL;
  VMZeroTimePa : TIME;
  VMMinDTimePa : TIME;
  SynchPOCStInit : BOOL;
END_STRUCT;
END_TYPE

TYPE Sync_In : STRUCT
  CloseCmd : BOOL;
  OpenCmd : BOOL;
END_STRUCT;
END_TYPE

TYPE Synch_Out : STRUCT
  Ready : BOOL;
  Alarm : BOOL;
  CmdUPf : BOOL;
  CmdDNf : BOOL;
  CmdUPV : BOOL;
  CmdDNV : BOOL;
  SyncCheckSt : BOOL;
END_STRUCT;
END_TYPE

TYPE Synch_Struct : STRUCT
  Synch_Parameters : Synch_Parameters;
  Synch_Out : Synch_Out;
  Sync_In : Sync_In;
END_STRUCT;
END_TYPE

TYPE Synch_Dat : ARRAY[1..2] OF Synch_Parameters;
END_TYPE

TYPE InBattPLCLogic : STRUCT
  WD_QueryVal : UINT;
  Send_WD_Cmd : BOOL;
  BmsSys : BMS_Sys;
  ExtReadySt : BOOL;
  BattPLCParamStruct : BattPLCParamStruct;
  Batt_DisableCmd : BOOL;
  Batt_EnableCmd : BOOL;
  Batt_AlResetCmd : BOOL;
  FireAl : BOOL;
  EStop : BOOL;
  BMSMbCtrlStructIn : MbCtrlStruct;
  BmsRack : BMS_RackArray;
  Send_ClockSyncCmd : BOOL;
END_STRUCT;
END_TYPE

TYPE OutBattPLCLogic : STRUCT
  BMSMbCtrlStructOut : MbCtrlStruct;
  Batt_Bank : Batt_Bank_Array;
  Batt_Rack : Batt_Rack;
  Batt_Sys : Batt_Sys;
END_STRUCT;
END_TYPE

TYPE InBattPLCModbus : STRUCT
  ssMethodType : SINT;
  FSet : REAL;
  FAct : REAL;
END_STRUCT;
END_TYPE

TYPE OutBattPLCModbus : STRUCT
  ssMethodType : SINT;
  FSet : REAL;
  FAct : REAL;
END_STRUCT;
END_TYPE

TYPE BattPLCParameters : STRUCT
  MbCommTOutPa : TIME;
  MessageTimeDelayPa : TIME;
  NbOfRackPa : INT;
  NbOfBankPa : INT;
  MapOfRackPa : MapOfRackStruct;
  InvDcBusUMinPa : REAL;
  BattSysSyncUBiasPa : REAL;
  InvDcBusUMaxPa : REAL;
  BattRackNomEActPa : REAL;
  BattRackNomPActPa : REAL;
  InvPActMinPa : REAL;
  InvPActMaxPa : REAL;
  MinPctOfRkPa : REAL;
  RacksStartingTimeoutPa : TIME;
  Batt_SYSSyncRangePa : REAL;
  DrtChrgOnSocLookUpSocPa : DerateLookUpPa;
  DrtChrgOnSocLookUpDrtPa : DerateLookUpPa;
  DrtDChrgOnSocLookUpSocPa : DerateLookUpPa;
  DrtDChrgOnSocLookUpDrtPa : DerateLookUpPa;
  DerateTempLookUpTempPa : DerateLookUpPa;
  DerateTempLookUpDeratePa : DerateLookUpPa;
  RacksStoppingTimeoutPa : TIME;
  EnDerateWrtSocPa : BOOL;
  EnDerateWrtTempPa : BOOL;
  ClockSyncIntervalPa : TIME;
  WatchDogModePa : INT;
  ClockSyncEnPA : BOOL;
END_STRUCT;
END_TYPE

TYPE BattPLCParameters_Array : ARRAY[0..10] OF BattPLCParameters;
END_TYPE

TYPE BattPLCLogic : STRUCT
  In : InBattPLCLogic;
  Out : OutBattPLCLogic;
END_STRUCT;
END_TYPE

TYPE BattPLCLogic_Array : ARRAY[0..10] OF BattPLCLogic;
END_TYPE

TYPE BattPLCModbus : STRUCT
  In : InBattPLCModbus;
  Out : OutBattPLCModbus;
END_STRUCT;
END_TYPE

TYPE BattPLCModbus_Array : ARRAY[0..10] OF BattPLCModbus;
END_TYPE

TYPE emC_BattPLC : STRUCT
  CtrlLo : BattPLCLogic;
  Modbus : BattPLCModbus;
  Pa : BattPLCParameters;
END_STRUCT;
END_TYPE

TYPE emC_Ps_SMIn : STRUCT
  SSMethodType : SINT;
  ManualSt : BOOL;
  OperatorCmd : BOOL;
  AutoCmd : BOOL;
  OnlineSt : BOOL;
  RunningSt : BOOL;
  HealthySt : BOOL;
  BatReadySt : BOOL;
  BatOnlineSt : BOOL;
  BatEmergencyStop : BOOL;
  OpStartCmd : BOOL;
  OpStopCmd : BOOL;
  AutoStartCmd : BOOL;
  AutoStopCmd : BOOL;
  SchedulerStartStopCmd : BOOL;
  ResetCmd : BOOL;
  BatForceStop : BOOL;
  StopRampSt : BOOL;
  CriticalAlarm : BOOL;
  NonCriticalAlarm : BOOL;
  Warning : BOOL;
  AmILastGfm : BOOL;
  Timestamp : STRING(80);
  StartStopEnablePa : BOOL;
  StartingTimePa : TIME;
  StoppingTimePa : TIME;
  CoolingTimePa : TIME;
  MinRunTimePa : TIME;
  CmdOutTimePa : TIME;
  BatStartingTimePa : TIME;
  BatStoppingTimePa : TIME;
  SchedulerStartStopCmdEnPa : BOOL;
  LogDisPa : BOOL;
  ClearLogEnPa : BOOL;
END_STRUCT;
END_TYPE

TYPE emC_Ps_SMOut : STRUCT
  ManualMd : BOOL;
  OperatorMd : BOOL;
  AutoMd : BOOL;
  StartingSt : BOOL;
  StoppingSt : BOOL;
  BatStartingSt : BOOL;
  BatStoppingSt : BOOL;
  CoolingTimeActiveSt : BOOL;
  MinRunTimeActiveSt : BOOL;
  FailedToStartAl : BOOL;
  FailedToStopAl : BOOL;
  GcStartCmdOut : BOOL;
  GcStopCmdOut : BOOL;
  GcStartStopCmdOut : BOOL;
  BatEnCmdOut : BOOL;
  BatDisCmdOut : BOOL;
  BatEnDisCmdOut : BOOL;
  SchedulableSt : BOOL;
  UnPSStartStopAlarm : BOOL;
  ExtInt : ExtIntESM;
  SMLog : emCSMLog;
END_STRUCT;
END_TYPE

TYPE emC_PsStateMachine : STRUCT
  In : emC_Ps_SMIn;
  Out : emC_Ps_SMOut;
END_STRUCT;
END_TYPE

TYPE emPsIn_In : STRUCT
  SSMethodType : SINT;
  PS_Out_EXTINT : PS_Out_EXTINT;
END_STRUCT;
END_TYPE

TYPE emPsIn_Out : STRUCT
  PSisNotResponding : BOOL;
  PSisResponding : BOOL;
  ExceptionFromSlave : BOOL;
  PS_In_EXTINT : PS_In_EXTINT;
END_STRUCT;
END_TYPE

TYPE emPsInDT : STRUCT
  In : emPsIn_In;
  Out : emPsIn_Out;
END_STRUCT;
END_TYPE

TYPE emPsOut_In : STRUCT
  SSMethodType : SINT;
  FSetOut : REAL;
  USetOut : REAL;
  PSetOut : REAL;
  QSetOut : REAL;
  BlackSys : BOOL;
  NetOnlineSt : BOOL;
  NetIslandReq : BOOL;
  ExtInt : ExtIntESM;
  PmLostComms : BOOL;
  FNomPa : REAL;
  UNomPa : REAL;
  PQFVSelPaGfw : BOOL;
  PQFVSelPaGfm : BOOL;
  PLimMaxPa : REAL;
  PLimMinPa : REAL;
  QLimMaxPa : REAL;
  QLimMinPa : REAL;
  AllowGFWEnPa : BOOL;
  AllowGFMEnPa : BOOL;
  InvertHwEnablePa : BOOL;
  PhaseRotationPa : BOOL;
  FastSlowDataEnPa : BOOL;
  SelModMapPa : INT;
  PS_In_EXTINT : PS_In_EXTINT;
END_STRUCT;
END_TYPE

TYPE emPsOut_Out : STRUCT
  PS_Out_EXTINT : PS_Out_EXTINT;
  GridFormingSel : BOOL;
END_STRUCT;
END_TYPE

TYPE emPsOutDT : STRUCT
  In : emPsOut_In;
  Out : emPsOut_Out;
END_STRUCT;
END_TYPE

TYPE emPsDT : STRUCT
  PS : PS;
  emPsIn : emPsInDT;
  emPsOut : emPsOutDT;
END_STRUCT;
END_TYPE

TYPE MSHIn : STRUCT
  ManualSt : BOOL;
  CriticalAlarm : BOOL;
  NonCriticalAlarm : BOOL;
  Warning : BOOL;
END_STRUCT;
END_TYPE

TYPE MSHOut : STRUCT
  Example : BOOL;
END_STRUCT;
END_TYPE

TYPE Field : STRUCT
  MSHIn : MSHIn;
  MSHOut : MSHOut;
END_STRUCT;
END_TYPE

TYPE emC_Ps_SCADAIn : STRUCT
  StartCmd : BOOL;
  StopCmd : BOOL;
  AlarmReset : BOOL;
  BreakerOpen : BOOL;
  BreakerClose : BOOL;
  ExtSetEnSt : BOOL;
  BlackOutResCmd : BOOL;
  PSet : REAL;
  QSet : REAL;
  USet : REAL;
  FSet : REAL;
END_STRUCT;
END_TYPE

TYPE RkSCADAOut : STRUCT
  OnlineSt : BOOL;
  FaultSt : BOOL;
  SoCAct : REAL;
  SoHAct : REAL;
  UAct : REAL;
  IAct : REAL;
  TempAct : REAL;
END_STRUCT;
END_TYPE

TYPE Rk : ARRAY[1..32] OF RkSCADAOut;
END_TYPE

TYPE emC_Ps_SCADAOut : STRUCT
  U12Act : REAL;
  U23Act : REAL;
  U31Act : REAL;
  IAvgAct : REAL;
  I1Act : REAL;
  I2Act : REAL;
  I3Act : REAL;
  PfAct : REAL;
  BatSyncUAct : REAL;
  BatSocAct : REAL;
  TempAct : REAL;
  UAct : REAL;
  PAct : REAL;
  QAct : REAL;
  EAct : REAL;
  FAct : REAL;
  GcSPNomAct : REAL;
  GcINomAct : REAL;
  GcUNomAct : REAL;
  GcFNomAct : REAL;
  GcModUNomAct : REAL;
  OperatorMd : BOOL;
  AutoMd : BOOL;
  LocalOnlineSt : BOOL;
  ManualMd : BOOL;
  FailedToStartAl : BOOL;
  FailedToStopAl : BOOL;
  NonCriticalAl : BOOL;
  WarningAl : BOOL;
  CriticalAl : BOOL;
  EstopAl : BOOL;
  FaultAl : BOOL;
  HealthySt : BOOL;
  OnlineSt : BOOL;
  RunningSt : BOOL;
  BatEmergencyStop : BOOL;
  BlackOutCondition : BOOL;
  BatInitializeSt : BOOL;
  BatNotReadySt : BOOL;
  BatReadySt : BOOL;
  BatStartingSt : BOOL;
  BatOnlineSt : BOOL;
  BatStoppingSt : BOOL;
  BmsVersion : REAL;
  BmsRacksNServiceCnt : REAL;
  BmsTotalRackCnt : REAL;
  BmsHeartBeat : REAL;
  BmsPartMinRackCnt : REAL;
  BmsPartDiffVolt : REAL;
  BmsEStopProtEn : BOOL;
  BmsEStopSPDEn : BOOL;
  BmsChargingSt : BOOL;
  BmsDischargingSt : BOOL;
  BattRunningSt : BOOL;
  BmsRkPartOnlineSt : BOOL;
  BmsEStopSPDSt : BOOL;
  BmsEStopProtSt : BOOL;
  BmsEStopPartSt : BOOL;
  BmsHealthySt : BOOL;
  BmsFireSysOkSt : BOOL;
  BmsCriticalAl : BOOL;
  BmsNonCriticalAl : BOOL;
  BmsWarningAl : BOOL;
  BmsStateTOUT : BOOL;
  BmsInitCommsFail : BOOL;
  BmsMinRkCloseFail : BOOL;
  BmsRkTripStart : BOOL;
  BmsMinRkOnlineFail : BOOL;
  BmsRkFailToOpen : BOOL;
  BmsSysFireAl : BOOL;
  BmsBmsLostCommsAl : BOOL;
  BmsBankFault : BOOL;
  BmsEStopAl : BOOL;
  BmsExtReadyStNotSetAl : BOOL;
  BattUSyncErrAl : BOOL;
  BmsRkFail2Cls : BOOL;
  BmsRkCntrFailAl : BOOL;
  BmsRTUComAl : BOOL;
  BmsRTUComFlt : BOOL;
  BmsRkVoltImbAl : BOOL;
  BmsSysStopAl : BOOL;
  BmsModuleUnderTempAl : BOOL;
  BmsModuleOverTempAl : BOOL;
  BmsModuleUnVoltAl : BOOL;
  BmsModuleOvVoltAl : BOOL;
  BmsRackVoltRegAl : BOOL;
  BmsRackTempRegAl : BOOL;
  BmsAuxProtAl : BOOL;
  BmsChargeOperLimAl : BOOL;
  BmsDischargeOperLimAl : BOOL;
  BmsRackUnVoltAl : BOOL;
  BmsRackOvVoltAl : BOOL;
  BmsRackCommsAl : BOOL;
  BmsTrayCommsAl : BOOL;
  BmsDcCntrSensor1Al : BOOL;
  BmsDcCntrSensor2Al : BOOL;
  BmsFanFailAl : BOOL;
  BmsChargeOverCurrentAl : BOOL;
  BmsDisChargeOverCurrentAl : BOOL;
  BmsRackVSenseDiffAl : BOOL;
  BmsRackFuseFailAl : BOOL;
  BmsRackCurrentSenserFailAl : BOOL;
  BmsRackPermanentUVAl : BOOL;
  BmsDcCntr1Al : BOOL;
  BmsDcCntr2Al : BOOL;
  BmsDcSwCntFailAl : BOOL;
  BmsCellVoltSenFailAl : BOOL;
  BmsDCFuseSenserFailAl : BOOL;
  BmsModuleUnderTempProt : BOOL;
  BmsModuleOverTempProt : BOOL;
  BmsModuleUnVoltProt : BOOL;
  BmsModuleOvVoltProt : BOOL;
  BmsRackVoltRegProt : BOOL;
  BmsRackTempRegProt : BOOL;
  BmsAuxProtProt : BOOL;
  BmsChargeOperLimProt : BOOL;
  BmsDischargeOperLimProt : BOOL;
  BmsRackUnVoltProt : BOOL;
  BmsRackOvVoltProt : BOOL;
  BmsRackCommsProt : BOOL;
  BmsTrayCommsProt : BOOL;
  BmsDcCntrSensor1Prot : BOOL;
  BmsDcCntrSensor2Prot : BOOL;
  BmsFanFailProt : BOOL;
  BmsChargeOverCurrentProt : BOOL;
  BmsDisChargeOverCurrentProt : BOOL;
  BmsRackVSenseDiffProt : BOOL;
  BmsRackFuseFailProt : BOOL;
  BmsRackCurrentSenserFailProt : BOOL;
  BmsRackPermanentUVProt : BOOL;
  BmsDcCntr1Prot : BOOL;
  BmsDcCntr2Prot : BOOL;
  BmsDcSwCntFailProt : BOOL;
  BmsCellVoltSenFailProt : BOOL;
  BmsDCFuseSenserFailProt : BOOL;
  BmsUdcAct : REAL;
  BmsIdcAct : REAL;
  BmsNomPAct : REAL;
  BmsNomEAct : REAL;
  BatPNomMaxAct : REAL;
  BatPNomMinAct : REAL;
  BmsPAct : REAL;
  BmsEAct : REAL;
  BmsSocPctAct : REAL;
  BmsSohAct : REAL;
  BmsTempMaxAct : REAL;
  BmsTempMinAct : REAL;
  BmsSyncUSet : REAL;
  Rk : Rk;
  GCRunningSt : BOOL;
  GCHealthy : BOOL;
  GCStartingSt : BOOL;
  GCReadySt : BOOL;
  GCGridFollowing : BOOL;
  GCFaultSt : BOOL;
  GCGridForming : BOOL;
  GCAreaEPSLost : BOOL;
  GCChargingSt : BOOL;
  GCRideThru : BOOL;
  GCTransitionActiveSt : BOOL;
  GCGndFault : BOOL;
  GCDCOverU : BOOL;
  GCACDisconnect : BOOL;
  GCDCDisconnect : BOOL;
  GCDCGridDisconnect : BOOL;
  GCCabinetOpen : BOOL;
  GCManualShutdown : BOOL;
  GCOverTemp : BOOL;
  GCOverF : BOOL;
  GCUnderF : BOOL;
  GCACOverVolt : BOOL;
  GCACUnderVolt : BOOL;
  GCBlownFuse : BOOL;
  GCUnderTemp : BOOL;
  GCMemLoss : BOOL;
  GCHWTestFailed : BOOL;
  PSStateWord : REAL;
  GCPAct : REAL;
  GCFAct : REAL;
  GCSNomAct : REAL;
  GCQAct : REAL;
  GCPF : REAL;
  GCEAct : REAL;
  GCTempAct : REAL;
  GCIGBTTempaAct : REAL;
  GCTrafoTempAct : REAL;
  GCOTTempAct : REAL;
  GCUAct12 : REAL;
  GCUAct23 : REAL;
  GCUAct13 : REAL;
  GCUAct1N : REAL;
  GCUAct2N : REAL;
  GCUAct3N : REAL;
  GCUAct : REAL;
  GCABBCtrlWrongConfig : BOOL;
  GCABBCtrlReady : BOOL;
  GCABBCtrlStartingSt : BOOL;
  GCABBCtrlVGMActiveSt : BOOL;
  GCABBCtrlGSMActiveSt : BOOL;
  GCABBCtrlError : BOOL;
  GCABBCtrlStoppingSt : BOOL;
  GCABBCtrlIslanded : BOOL;
  GCABBStateWord : REAL;
  GCABBErrorID : REAL;
  GCLostComms : BOOL;
  GCCommsOk : BOOL;
  GCHardwareenablestatus : BOOL;
  GCACPowerAvailable : BOOL;
  GCDCPowerAvailable : BOOL;
  GCPowerCircuitEnabled : BOOL;
  GCMX1relaystatus : BOOL;
  GCMX2relaystatus : BOOL;
  GCPrechargestatus : BOOL;
  GCK2Relaystatus : BOOL;
  GCControlcommandsvalid : BOOL;
  GCPowercommandValid : BOOL;
  GCCurrentcommandValid : BOOL;
  GCPhaserotationstatus : BOOL;
  GCLinevoltagedetected : BOOL;
  GCUnused : BOOL;
  GCRemoteACPowerAvailable : BOOL;
  GCRemotephaserotationstatus : BOOL;
  GCRemoteLineVoltageDetected : BOOL;
  GCDI1Status : BOOL;
  GCDI2Status : BOOL;
  GCDI3Status : BOOL;
  GCDI4Status : BOOL;
  GCDO1Status : BOOL;
  GCDO2Status : BOOL;
  GCDO3Status : BOOL;
  GCDO4Status : BOOL;
  GCDClinkRefCmdValid : BOOL;
  GCPumpRunning : BOOL;
  GCPumpFault : BOOL;
  GCABBLostCommsStop : BOOL;
  GCCtrlSystemReady : BOOL;
  GCSysFltCode : REAL;
  GCFlt_Estp : BOOL;
  GCFlt_ACOverCurrent : BOOL;
  GCFlt_DCOverCurrent : BOOL;
  GCFlt_DCOverVoltage : BOOL;
  GCFlt_PDOverTemp : BOOL;
  GCFlt_InvOverTemp : BOOL;
  GCFlt_CmdMsg : BOOL;
  GCFlt_DCUnderVolt : BOOL;
  GCFlt_ACOverVolt : BOOL;
  GCFlt_IllegalTrans : BOOL;
  GCFlt_EEHeat : BOOL;
  GCFlt_EESction : BOOL;
  GCFlt_Cool : BOOL;
  GCFlt_TimedOverLoadAC : BOOL;
  GCFlt_TimedOverLoadDC : BOOL;
  GCFlt_ICOL : BOOL;
  GCFlt_CtlBdVolt : BOOL;
  GCFlt_PChImbal : BOOL;
  GCFlt_DiDt : BOOL;
  GCFlt_CoolingFlw : BOOL;
  GCFlt_ThrmOverLoad : BOOL;
  GCFlt_Fan : BOOL;
  GCFlt_POR : BOOL;
  GCFlt_Condensation : BOOL;
  GCFlt_I2C : BOOL;
  GCFlt_ExternalInhibit : BOOL;
  GCFlt_GroundFault : BOOL;
  GCFlt_Fuse : BOOL;
  GCFlt_Rsvd28 : BOOL;
  GCFlt_ACDisconnect : BOOL;
  GCFlt_Rsvd30 : BOOL;
  GCFlt_Rsvd31 : BOOL;
  GCWrn_CANW : BOOL;
  GCWrn_CANEP : BOOL;
  GCWrn_Thrm : BOOL;
  GCWrn_Fan : BOOL;
  GCWrn_EeSaveActive : BOOL;
  GCWrn_LocNetMismatch : BOOL;
  GCWrn_RemNetMismatch : BOOL;
  GCWrn_Condensation : BOOL;
  GCWrn_I2C : BOOL;
  GCWrn_ExternalInhibit : BOOL;
  GCWrn_MaintReqd : BOOL;
  GCWrn_GroundFault : BOOL;
  GCWrn_Fuse : BOOL;
  GCWrn_ACDisconnect : BOOL;
  GCWrn_Rsvd14 : BOOL;
  GCWrn_Rsvd15 : BOOL;
  GCWrn_Rsvd16 : BOOL;
  GCWrn_Rsvd17 : BOOL;
  GCWrn_Rsvd18 : BOOL;
  GCWrn_Rsvd19 : BOOL;
  GCWrn_Rsvd20 : BOOL;
  GCWrn_Rsvd21 : BOOL;
  GCWrn_Rsvd22 : BOOL;
  GCWrn_Rsvd23 : BOOL;
  GCWrn_Rsvd24 : BOOL;
  GCWrn_Rsvd25 : BOOL;
  GCWrn_Rsvd26 : BOOL;
  GCWrn_Rsvd27 : BOOL;
  GCWrn_Rsvd28 : BOOL;
  GCWrn_Rsvd29 : BOOL;
  GCWrn_Rsvd30 : BOOL;
  GCCriticalAlarm : BOOL;
  GCNonCriticalAlarm : BOOL;
  GCWarning : BOOL;
  GCreconnectDelay : BOOL;
  GCMomentCessation : BOOL;
  GCInhibited : BOOL;
END_STRUCT;
END_TYPE

TYPE emC_PsSCADA : STRUCT
  In : emC_Ps_SCADAIn;
  Out : emC_Ps_SCADAOut;
END_STRUCT;
END_TYPE

TYPE LuC_PPCIn_Out : STRUCT
  FSetOut : REAL;
  USetOut : REAL;
  PSetOut : REAL;
  QSetOut : REAL;
  NetOnlineSt : BOOL;
  NetIslandReq : BOOL;
  AutoStartCmd : BOOL;
  AutoStopCmd : BOOL;
  StopRampSt : BOOL;
END_STRUCT;
END_TYPE

TYPE LuC_PPCIn_In : STRUCT
  SetPointRampEnPa : BOOL;
  FSetOutRmpUpPa : REAL;
  FSetOutRmpDownPa : REAL;
  USetOutRmpUpPa : REAL;
  USetOutRmpDownPa : REAL;
  PSetOutRmpUpPa : REAL;
  PSetOutRmpDownPa : REAL;
  QSetOutRmpUpPa : REAL;
  QSetOutRmpDownPa : REAL;
END_STRUCT;
END_TYPE

TYPE LuC_PPCIn : STRUCT
  In : LuC_PPCIn_In;
  Out : LuC_PPCIn_Out;
END_STRUCT;
END_TYPE

TYPE LuC_PPCOut : STRUCT
  GCFaultSt : BOOL;
  TempAct : REAL;
  OnlineSt : BOOL;
  RunningSt : BOOL;
  NonCriticalAlarm : BOOL;
  CriticalAlarm : BOOL;
  Warning : BOOL;
  StoppingSt : BOOL;
  BatPNomMaxAct : REAL;
  BatPNomMinAct : REAL;
  SocPctAct : REAL;
  UAct : REAL;
  FAct : REAL;
  PAct : REAL;
  QAct : REAL;
  CtrlSystemReady : BOOL;
  BlackSys : BOOL;
END_STRUCT;
END_TYPE

TYPE LuC_PPC : STRUCT
  PPCIn : LuC_PPCIn;
  PPCOut : LuC_PPCOut;
END_STRUCT;
END_TYPE

TYPE LUC_BESS_Parameters_In : STRUCT
  PCtrlDeadbPa : REAL;
  PLimMaxPa : REAL;
  PLimMinPa : REAL;
  P_StoprampDownPa : REAL;
  P_StoprampUpPa : REAL;
  QCtrlDeadbPa : REAL;
  QLimMaxPa : REAL;
  QLimMinPa : REAL;
  Q_StoprampDownPa : REAL;
  Q_StoprampUpPa : REAL;
END_STRUCT;
END_TYPE

TYPE LUC_BESS_Logic_In : STRUCT
  ssMethodType : SINT;
  StoppingSt : BOOL;
  PAct : REAL;
  QAct : REAL;
END_STRUCT;
END_TYPE

TYPE LUC_BESS_Logic_Out : STRUCT
  PLimmaxPa : REAL;
  PLimminPa : REAL;
  QLimmaxPa : REAL;
  QLimminPa : REAL;
  StopRampSt : BOOL;
END_STRUCT;
END_TYPE

TYPE LUC_BESS_Logic : STRUCT
  In : LUC_BESS_Logic_In;
  Out : LUC_BESS_Logic_Out;
END_STRUCT;
END_TYPE

TYPE emC_LUC_Ctrl : STRUCT
  LUC_BESS_Parameters : LUC_BESS_Parameters_In;
  LUC_BESS_Logic : LUC_BESS_Logic;
END_STRUCT;
END_TYPE

TYPE emC_LUC : STRUCT
  Field : Field;
  emPs : emPsDT;
  BattPLC : emC_BattPLC;
  SM : emC_PsStateMachine;
  SCADA : emC_PsSCADA;
  emC_LUC_Ctrl : emC_LUC_Ctrl;
  PPC : LuC_PPC;
END_STRUCT;
END_TYPE

TYPE emC_LUC_Array : ARRAY[1..5] OF emC_LUC;
END_TYPE

TYPE PPC_LuCOut : STRUCT
  FSetOut : REAL;
  USetOut : REAL;
  PSetOut : REAL;
  QSetOut : REAL;
  F_SF : REAL;
  U_SF : REAL;
  P_SF : REAL;
  Q_SF : REAL;
  NetOnlineSt : BOOL;
  NetIslandReq : BOOL;
  AutoStartCmd : BOOL;
  AutoStopCmd : BOOL;
  StopRampSt : BOOL;
  BlackSys : BOOL;
END_STRUCT;
END_TYPE

TYPE PPC_LuCIn : STRUCT
  ComFault : BOOL;
  GCFaultSt : BOOL;
  TempAct : REAL;
  OnlineSt : BOOL;
  RunningSt : BOOL;
  NonCriticalAlarm : BOOL;
  CriticalAlarm : BOOL;
  Warning : BOOL;
  StoppingSt : BOOL;
  BatPNomMaxAct : REAL;
  BatPNomMinAct : REAL;
  SocPctAct : REAL;
  UAct : REAL;
  FAct : REAL;
  PAct : REAL;
  QAct : REAL;
  CtrlSystemReady : BOOL;
  BlackSys : BOOL;
END_STRUCT;
END_TYPE

TYPE PPC_Param : STRUCT
  NbOfLuCPa : INT;
  FastSlowDataEnPa : BOOL;
  PQFVSelPaGfw : BOOL;
  PQFVSelPaGfm : BOOL;
  AllowGFWEnPa : BOOL;
  AllowGFMEnPa : BOOL;
END_STRUCT;
END_TYPE

TYPE PPC_Summary : STRUCT
  GCFaultSt : BOOL;
  AvgTempAct : REAL;
  OnlineSt : BOOL;
  RunningSt : BOOL;
  NonCriticalAlarm : BOOL;
  CriticalAlarm : BOOL;
  Warning : BOOL;
  StoppingSt : BOOL;
  TotBatPNomMaxAct : REAL;
  TotBatPNomMinAct : REAL;
  AvgSocPct : REAL;
  AvgUAct : REAL;
  AvgFAct : REAL;
  TotPAct : REAL;
  TotQAct : REAL;
  BlackSys : BOOL;
  ComFaultCnt : INT;
  OnlineCnt : INT;
END_STRUCT;
END_TYPE

TYPE PPC_LuC : STRUCT
  In : PPC_LuCIn;
  Out : PPC_LuCOut;
END_STRUCT;
END_TYPE

TYPE PPC_Luc_Array : ARRAY[1..32] OF PPC_LuC;
END_TYPE

TYPE emC_PPC : STRUCT
  LuC : PPC_Luc_Array;
  Summary : PPC_Summary;
  Param : PPC_Param;
END_STRUCT;
END_TYPE

TYPE emC_PPC_Array : ARRAY[1..4] OF emC_PPC;
END_TYPE

PROGRAM emC_PPC_R01_MSH_In
  VAR_EXTERNAL
    emC_PPC : emC_PPC_Array;
    PPCNum : INT;
  END_VAR
  VAR
    emC_PPC_LuCIn_1 : emC_PPC_LuCIn;
    emC_PPC_LuCIn_2 : emC_PPC_LuCIn;
    emC_PPC_LuCIn_3 : emC_PPC_LuCIn;
    emC_PPC_LuCIn_4 : emC_PPC_LuCIn;
    emC_PPC_LuCIn_5 : emC_PPC_LuCIn;
  END_VAR
  VAR_EXTERNAL
    LuCNum : INT;
  END_VAR
  VAR
    NbOfLuCPa_S : INT := 2;
    FastSlowDataEnPa_S : BOOL := 0;
    AllowGFMEnPa_S : BOOL;
    AllowGFWEnPa_S : BOOL;
    PQFVSelPaGfm_S : BOOL;
    PQFVSelPaGfw_S : BOOL;
    L1_GCFaultSt_I : SPI;
    L1_NonCriticalAlarm_I : SPI;
    L1_CriticalAlarm_I : SPI;
    L1_Warning_I : SPI;
    L1_StoppingSt_I : SPI;
    L1_CtrlSystemReady_I : SPI;
    L1_BlackSys_I : SPI;
    L1_BatPNomMaxAct_I : MFI;
    L1_BatPNomMinAct_I : MFI;
    L1_SocPctAct_I : MFI;
    L1_UAct_I : MFI;
    L1_FAct_I : MFI;
    L1_PAct_I : MFI;
    L1_QAct_I : MFI;
    L1_TempAct_I : MFI;
    L1_Inoperable_I : SEV;
    L1_OnlineSt_I : SPI;
    L1_RunningSt_I : SPI;
    L2_GCFaultSt_I : SPI;
    L2_NonCriticalAlarm_I : SPI;
    L2_CriticalAlarm_I : SPI;
    L2_Warning_I : SPI;
    L2_StoppingSt_I : SPI;
    L2_CtrlSystemReady_I : SPI;
    L2_BlackSys_I : SPI;
    L2_BatPNomMaxAct_I : MFI;
    L2_BatPNomMinAct_I : MFI;
    L2_SocPctAct_I : MFI;
    L2_UAct_I : MFI;
    L2_FAct_I : MFI;
    L2_PAct_I : MFI;
    L2_QAct_I : MFI;
    L2_TempAct_I : MFI;
    L2_Inoperable_I : SEV;
    L2_OnlineSt_I : SPI;
    L2_RunningSt_I : SPI;
    L3_GCFaultSt_I : SPI;
    L3_NonCriticalAlarm_I : SPI;
    L3_CriticalAlarm_I : SPI;
    L3_Warning_I : SPI;
    L3_StoppingSt_I : SPI;
    L3_CtrlSystemReady_I : SPI;
    L3_BlackSys_I : SPI;
    L3_BatPNomMaxAct_I : MFI;
    L3_BatPNomMinAct_I : MFI;
    L3_SocPctAct_I : MFI;
    L3_UAct_I : MFI;
    L3_FAct_I : MFI;
    L3_PAct_I : MFI;
    L3_QAct_I : MFI;
    L3_TempAct_I : MFI;
    L3_Inoperable_I : SEV;
    L3_OnlineSt_I : SPI;
    L3_RunningSt_I : SPI;
    L4_GCFaultSt_I : SPI;
    L4_NonCriticalAlarm_I : SPI;
    L4_CriticalAlarm_I : SPI;
    L4_Warning_I : SPI;
    L4_StoppingSt_I : SPI;
    L4_CtrlSystemReady_I : SPI;
    L4_BlackSys_I : SPI;
    L4_BatPNomMaxAct_I : MFI;
    L4_BatPNomMinAct_I : MFI;
    L4_SocPctAct_I : MFI;
    L4_UAct_I : MFI;
    L4_FAct_I : MFI;
    L4_PAct_I : MFI;
    L4_QAct_I : MFI;
    L4_TempAct_I : MFI;
    L4_Inoperable_I : SEV;
    L4_OnlineSt_I : SPI;
    L4_RunningSt_I : SPI;
    L5_GCFaultSt_I : SPI;
    L5_NonCriticalAlarm_I : SPI;
    L5_CriticalAlarm_I : SPI;
    L5_Warning_I : SPI;
    L5_StoppingSt_I : SPI;
    L5_CtrlSystemReady_I : SPI;
    L5_BlackSys_I : SPI;
    L5_BatPNomMaxAct_I : MFI;
    L5_BatPNomMinAct_I : MFI;
    L5_SocPctAct_I : MFI;
    L5_UAct_I : MFI;
    L5_FAct_I : MFI;
    L5_PAct_I : MFI;
    L5_QAct_I : MFI;
    L5_TempAct_I : MFI;
    L5_Inoperable_I : SEV;
    L5_OnlineSt_I : SPI;
    L5_RunningSt_I : SPI;
  END_VAR

						
							(*NbOfLuCPa	:=	2	;*)
LuCNum	:=	5	;
								
emC_PPC[PPCNum].Param.NbOfLuCPa	:=	NbOfLuCPa_S	;
PPCNum	:=	1	;
emC_PPC[PPCNum].Param.FastSlowDataEnPa	:=	FastSlowDataEnPa_S	;
emC_PPC[PPCNum].Param.AllowGFMEnPa	:=	AllowGFMEnPa_S	;
emC_PPC[PPCNum].Param.AllowGFWEnPa	:=	AllowGFWEnPa_S	;
emC_PPC[PPCNum].Param.PQFVSelPaGfm	:=	PQFVSelPaGfm_S	;
emC_PPC[PPCNum].Param.PQFVSelPaGfw	:=	PQFVSelPaGfw_S	;
							
							
							
							
								
emC_PPC_LuCIn_1(								
				GCFaultSt_I		:=	L1_GCFaultSt_I	,
				NonCriticalAlarm_I		:=	L1_NonCriticalAlarm_I	,
				CriticalAlarm_I		:=	L1_CriticalAlarm_I	,
				Warning_I		:=	L1_Warning_I	,
				StoppingSt_I		:=	L1_StoppingSt_I	,
				CtrlSystemReady_I		:=	L1_CtrlSystemReady_I	,
				BlackSys_I		:=	L1_BlackSys_I	,
				OnlineSt_I		:=	L1_OnlineSt_I	,
				RunningSt_I		:=	L1_RunningSt_I	,
				Inoperable_I		:=	L1_Inoperable_I	,
				BatPNomMaxAct_I		:=	L1_BatPNomMaxAct_I	,
				BatPNomMinAct_I		:=	L1_BatPNomMinAct_I	,
				SocPctAct_I		:=	L1_SocPctAct_I	,
				UAct_I		:=	L1_UAct_I	,
				FAct_I		:=	L1_FAct_I	,
				PAct_I		:=	L1_PAct_I	,
				QAct_I		:=	L1_QAct_I	,
				TempAct_I		:=	L1_TempAct_I	);
	emC_PPC[PPCNum].LuC[1].In.GCFaultSt	:=	emC_PPC_LuCIn_1.GCFaultSt	;				
	emC_PPC[PPCNum].LuC[1].In.NonCriticalAlarm	:=	emC_PPC_LuCIn_1.NonCriticalAlarm	;				
	emC_PPC[PPCNum].LuC[1].In.CriticalAlarm	:=	emC_PPC_LuCIn_1.CriticalAlarm	;				
	emC_PPC[PPCNum].LuC[1].In.Warning	:=	emC_PPC_LuCIn_1.Warning	;				
	emC_PPC[PPCNum].LuC[1].In.StoppingSt	:=	emC_PPC_LuCIn_1.StoppingSt	;				
	emC_PPC[PPCNum].LuC[1].In.CtrlSystemReady	:=	emC_PPC_LuCIn_1.CtrlSystemReady	;				
	emC_PPC[PPCNum].LuC[1].In.BlackSys	:=	emC_PPC_LuCIn_1.BlackSys	;				
	emC_PPC[PPCNum].LuC[1].In.OnlineSt	:=	emC_PPC_LuCIn_1.OnlineSt	;				
	emC_PPC[PPCNum].LuC[1].In.RunningSt	:=	emC_PPC_LuCIn_1.RunningSt	;				
	emC_PPC[PPCNum].LuC[1].In.ComFault	:=	emC_PPC_LuCIn_1.ComFault	;				
	emC_PPC[PPCNum].LuC[1].In.BatPNomMaxAct	:=	emC_PPC_LuCIn_1.BatPNomMaxAct	;				
	emC_PPC[PPCNum].LuC[1].In.BatPNomMinAct	:=	emC_PPC_LuCIn_1.BatPNomMinAct	;				
	emC_PPC[PPCNum].LuC[1].In.SocPctAct	:=	emC_PPC_LuCIn_1.SocPctAct	;				
	emC_PPC[PPCNum].LuC[1].In.UAct	:=	emC_PPC_LuCIn_1.UAct	;				
	emC_PPC[PPCNum].LuC[1].In.FAct	:=	emC_PPC_LuCIn_1.FAct	;				
	emC_PPC[PPCNum].LuC[1].In.PAct	:=	emC_PPC_LuCIn_1.PAct	;				
	emC_PPC[PPCNum].LuC[1].In.QAct	:=	emC_PPC_LuCIn_1.QAct	;				
	emC_PPC[PPCNum].LuC[1].In.TempAct	:=	emC_PPC_LuCIn_1.TempAct	;
							
							
								
emC_PPC_LuCIn_2(								
				GCFaultSt_I		:=	L2_GCFaultSt_I	,
				NonCriticalAlarm_I		:=	L2_NonCriticalAlarm_I	,
				CriticalAlarm_I		:=	L2_CriticalAlarm_I	,
				Warning_I		:=	L2_Warning_I	,
				StoppingSt_I		:=	L2_StoppingSt_I	,
				CtrlSystemReady_I		:=	L2_CtrlSystemReady_I	,
				BlackSys_I		:=	L2_BlackSys_I	,
				OnlineSt_I		:=	L2_OnlineSt_I	,
				RunningSt_I		:=	L2_RunningSt_I	,
				Inoperable_I		:=	L2_Inoperable_I	,
				BatPNomMaxAct_I		:=	L2_BatPNomMaxAct_I	,
				BatPNomMinAct_I		:=	L2_BatPNomMinAct_I	,
				SocPctAct_I		:=	L2_SocPctAct_I	,
				UAct_I		:=	L2_UAct_I	,
				FAct_I		:=	L2_FAct_I	,
				PAct_I		:=	L2_PAct_I	,
				QAct_I		:=	L2_QAct_I	,
				TempAct_I		:=	L2_TempAct_I	);
	emC_PPC[PPCNum].LuC[2].In.GCFaultSt	:=	emC_PPC_LuCIn_2.GCFaultSt	;				
	emC_PPC[PPCNum].LuC[2].In.NonCriticalAlarm	:=	emC_PPC_LuCIn_2.NonCriticalAlarm	;				
	emC_PPC[PPCNum].LuC[2].In.CriticalAlarm	:=	emC_PPC_LuCIn_2.CriticalAlarm	;				
	emC_PPC[PPCNum].LuC[2].In.Warning	:=	emC_PPC_LuCIn_2.Warning	;				
	emC_PPC[PPCNum].LuC[2].In.StoppingSt	:=	emC_PPC_LuCIn_2.StoppingSt	;				
	emC_PPC[PPCNum].LuC[2].In.CtrlSystemReady	:=	emC_PPC_LuCIn_2.CtrlSystemReady	;				
	emC_PPC[PPCNum].LuC[2].In.BlackSys	:=	emC_PPC_LuCIn_2.BlackSys	;				
	emC_PPC[PPCNum].LuC[2].In.OnlineSt	:=	emC_PPC_LuCIn_2.OnlineSt	;				
	emC_PPC[PPCNum].LuC[2].In.RunningSt	:=	emC_PPC_LuCIn_2.RunningSt	;				
	emC_PPC[PPCNum].LuC[2].In.ComFault	:=	emC_PPC_LuCIn_2.ComFault	;				
	emC_PPC[PPCNum].LuC[2].In.BatPNomMaxAct	:=	emC_PPC_LuCIn_2.BatPNomMaxAct	;				
	emC_PPC[PPCNum].LuC[2].In.BatPNomMinAct	:=	emC_PPC_LuCIn_2.BatPNomMinAct	;				
	emC_PPC[PPCNum].LuC[2].In.SocPctAct	:=	emC_PPC_LuCIn_2.SocPctAct	;				
	emC_PPC[PPCNum].LuC[2].In.UAct	:=	emC_PPC_LuCIn_2.UAct	;				
	emC_PPC[PPCNum].LuC[2].In.FAct	:=	emC_PPC_LuCIn_2.FAct	;				
	emC_PPC[PPCNum].LuC[2].In.PAct	:=	emC_PPC_LuCIn_2.PAct	;				
	emC_PPC[PPCNum].LuC[2].In.QAct	:=	emC_PPC_LuCIn_2.QAct	;				
	emC_PPC[PPCNum].LuC[2].In.TempAct	:=	emC_PPC_LuCIn_2.TempAct	;
							
							
								
emC_PPC_LuCIn_3(								
				GCFaultSt_I		:=	L3_GCFaultSt_I	,
				NonCriticalAlarm_I		:=	L3_NonCriticalAlarm_I	,
				CriticalAlarm_I		:=	L3_CriticalAlarm_I	,
				Warning_I		:=	L3_Warning_I	,
				StoppingSt_I		:=	L3_StoppingSt_I	,
				CtrlSystemReady_I		:=	L3_CtrlSystemReady_I	,
				BlackSys_I		:=	L3_BlackSys_I	,
				OnlineSt_I		:=	L3_OnlineSt_I	,
				RunningSt_I		:=	L3_RunningSt_I	,
				Inoperable_I		:=	L3_Inoperable_I	,
				BatPNomMaxAct_I		:=	L3_BatPNomMaxAct_I	,
				BatPNomMinAct_I		:=	L3_BatPNomMinAct_I	,
				SocPctAct_I		:=	L3_SocPctAct_I	,
				UAct_I		:=	L3_UAct_I	,
				FAct_I		:=	L3_FAct_I	,
				PAct_I		:=	L3_PAct_I	,
				QAct_I		:=	L3_QAct_I	,
				TempAct_I		:=	L3_TempAct_I	);
	emC_PPC[PPCNum].LuC[3].In.GCFaultSt	:=	emC_PPC_LuCIn_3.GCFaultSt	;				
	emC_PPC[PPCNum].LuC[3].In.NonCriticalAlarm	:=	emC_PPC_LuCIn_3.NonCriticalAlarm	;				
	emC_PPC[PPCNum].LuC[3].In.CriticalAlarm	:=	emC_PPC_LuCIn_3.CriticalAlarm	;				
	emC_PPC[PPCNum].LuC[3].In.Warning	:=	emC_PPC_LuCIn_3.Warning	;				
	emC_PPC[PPCNum].LuC[3].In.StoppingSt	:=	emC_PPC_LuCIn_3.StoppingSt	;				
	emC_PPC[PPCNum].LuC[3].In.CtrlSystemReady	:=	emC_PPC_LuCIn_3.CtrlSystemReady	;				
	emC_PPC[PPCNum].LuC[3].In.BlackSys	:=	emC_PPC_LuCIn_3.BlackSys	;				
	emC_PPC[PPCNum].LuC[3].In.OnlineSt	:=	emC_PPC_LuCIn_3.OnlineSt	;				
	emC_PPC[PPCNum].LuC[3].In.RunningSt	:=	emC_PPC_LuCIn_3.RunningSt	;				
	emC_PPC[PPCNum].LuC[3].In.ComFault	:=	emC_PPC_LuCIn_3.ComFault	;				
	emC_PPC[PPCNum].LuC[3].In.BatPNomMaxAct	:=	emC_PPC_LuCIn_3.BatPNomMaxAct	;				
	emC_PPC[PPCNum].LuC[3].In.BatPNomMinAct	:=	emC_PPC_LuCIn_3.BatPNomMinAct	;				
	emC_PPC[PPCNum].LuC[3].In.SocPctAct	:=	emC_PPC_LuCIn_3.SocPctAct	;				
	emC_PPC[PPCNum].LuC[3].In.UAct	:=	emC_PPC_LuCIn_3.UAct	;				
	emC_PPC[PPCNum].LuC[3].In.FAct	:=	emC_PPC_LuCIn_3.FAct	;				
	emC_PPC[PPCNum].LuC[3].In.PAct	:=	emC_PPC_LuCIn_3.PAct	;				
	emC_PPC[PPCNum].LuC[3].In.QAct	:=	emC_PPC_LuCIn_3.QAct	;				
	emC_PPC[PPCNum].LuC[3].In.TempAct	:=	emC_PPC_LuCIn_3.TempAct	;
							
							
								
emC_PPC_LuCIn_4(								
				GCFaultSt_I		:=	L4_GCFaultSt_I	,
				NonCriticalAlarm_I		:=	L4_NonCriticalAlarm_I	,
				CriticalAlarm_I		:=	L4_CriticalAlarm_I	,
				Warning_I		:=	L4_Warning_I	,
				StoppingSt_I		:=	L4_StoppingSt_I	,
				CtrlSystemReady_I		:=	L4_CtrlSystemReady_I	,
				BlackSys_I		:=	L4_BlackSys_I	,
				OnlineSt_I		:=	L4_OnlineSt_I	,
				RunningSt_I		:=	L4_RunningSt_I	,
				Inoperable_I		:=	L4_Inoperable_I	,
				BatPNomMaxAct_I		:=	L4_BatPNomMaxAct_I	,
				BatPNomMinAct_I		:=	L4_BatPNomMinAct_I	,
				SocPctAct_I		:=	L4_SocPctAct_I	,
				UAct_I		:=	L4_UAct_I	,
				FAct_I		:=	L4_FAct_I	,
				PAct_I		:=	L4_PAct_I	,
				QAct_I		:=	L4_QAct_I	,
				TempAct_I		:=	L4_TempAct_I	);
	emC_PPC[PPCNum].LuC[4].In.GCFaultSt	:=	emC_PPC_LuCIn_4.GCFaultSt	;				
	emC_PPC[PPCNum].LuC[4].In.NonCriticalAlarm	:=	emC_PPC_LuCIn_4.NonCriticalAlarm	;				
	emC_PPC[PPCNum].LuC[4].In.CriticalAlarm	:=	emC_PPC_LuCIn_4.CriticalAlarm	;				
	emC_PPC[PPCNum].LuC[4].In.Warning	:=	emC_PPC_LuCIn_4.Warning	;				
	emC_PPC[PPCNum].LuC[4].In.StoppingSt	:=	emC_PPC_LuCIn_4.StoppingSt	;				
	emC_PPC[PPCNum].LuC[4].In.CtrlSystemReady	:=	emC_PPC_LuCIn_4.CtrlSystemReady	;				
	emC_PPC[PPCNum].LuC[4].In.BlackSys	:=	emC_PPC_LuCIn_4.BlackSys	;				
	emC_PPC[PPCNum].LuC[4].In.OnlineSt	:=	emC_PPC_LuCIn_4.OnlineSt	;				
	emC_PPC[PPCNum].LuC[4].In.RunningSt	:=	emC_PPC_LuCIn_4.RunningSt	;				
	emC_PPC[PPCNum].LuC[4].In.ComFault	:=	emC_PPC_LuCIn_4.ComFault	;				
	emC_PPC[PPCNum].LuC[4].In.BatPNomMaxAct	:=	emC_PPC_LuCIn_4.BatPNomMaxAct	;				
	emC_PPC[PPCNum].LuC[4].In.BatPNomMinAct	:=	emC_PPC_LuCIn_4.BatPNomMinAct	;				
	emC_PPC[PPCNum].LuC[4].In.SocPctAct	:=	emC_PPC_LuCIn_4.SocPctAct	;				
	emC_PPC[PPCNum].LuC[4].In.UAct	:=	emC_PPC_LuCIn_4.UAct	;				
	emC_PPC[PPCNum].LuC[4].In.FAct	:=	emC_PPC_LuCIn_4.FAct	;				
	emC_PPC[PPCNum].LuC[4].In.PAct	:=	emC_PPC_LuCIn_4.PAct	;				
	emC_PPC[PPCNum].LuC[4].In.QAct	:=	emC_PPC_LuCIn_4.QAct	;				
	emC_PPC[PPCNum].LuC[4].In.TempAct	:=	emC_PPC_LuCIn_4.TempAct	;
							
							
								
emC_PPC_LuCIn_5(								
				GCFaultSt_I		:=	L5_GCFaultSt_I	,
				NonCriticalAlarm_I		:=	L5_NonCriticalAlarm_I	,
				CriticalAlarm_I		:=	L5_CriticalAlarm_I	,
				Warning_I		:=	L5_Warning_I	,
				StoppingSt_I		:=	L5_StoppingSt_I	,
				CtrlSystemReady_I		:=	L5_CtrlSystemReady_I	,
				BlackSys_I		:=	L5_BlackSys_I	,
				OnlineSt_I		:=	L5_OnlineSt_I	,
				RunningSt_I		:=	L5_RunningSt_I	,
				Inoperable_I		:=	L5_Inoperable_I	,
				BatPNomMaxAct_I		:=	L5_BatPNomMaxAct_I	,
				BatPNomMinAct_I		:=	L5_BatPNomMinAct_I	,
				SocPctAct_I		:=	L5_SocPctAct_I	,
				UAct_I		:=	L5_UAct_I	,
				FAct_I		:=	L5_FAct_I	,
				PAct_I		:=	L5_PAct_I	,
				QAct_I		:=	L5_QAct_I	,
				TempAct_I		:=	L5_TempAct_I	);
	emC_PPC[PPCNum].LuC[5].In.GCFaultSt	:=	emC_PPC_LuCIn_5.GCFaultSt	;				
	emC_PPC[PPCNum].LuC[5].In.NonCriticalAlarm	:=	emC_PPC_LuCIn_5.NonCriticalAlarm	;				
	emC_PPC[PPCNum].LuC[5].In.CriticalAlarm	:=	emC_PPC_LuCIn_5.CriticalAlarm	;				
	emC_PPC[PPCNum].LuC[5].In.Warning	:=	emC_PPC_LuCIn_5.Warning	;				
	emC_PPC[PPCNum].LuC[5].In.StoppingSt	:=	emC_PPC_LuCIn_5.StoppingSt	;				
	emC_PPC[PPCNum].LuC[5].In.CtrlSystemReady	:=	emC_PPC_LuCIn_5.CtrlSystemReady	;				
	emC_PPC[PPCNum].LuC[5].In.BlackSys	:=	emC_PPC_LuCIn_5.BlackSys	;				
	emC_PPC[PPCNum].LuC[5].In.OnlineSt	:=	emC_PPC_LuCIn_5.OnlineSt	;				
	emC_PPC[PPCNum].LuC[5].In.RunningSt	:=	emC_PPC_LuCIn_5.RunningSt	;				
	emC_PPC[PPCNum].LuC[5].In.ComFault	:=	emC_PPC_LuCIn_5.ComFault	;				
	emC_PPC[PPCNum].LuC[5].In.BatPNomMaxAct	:=	emC_PPC_LuCIn_5.BatPNomMaxAct	;				
	emC_PPC[PPCNum].LuC[5].In.BatPNomMinAct	:=	emC_PPC_LuCIn_5.BatPNomMinAct	;				
	emC_PPC[PPCNum].LuC[5].In.SocPctAct	:=	emC_PPC_LuCIn_5.SocPctAct	;				
	emC_PPC[PPCNum].LuC[5].In.UAct	:=	emC_PPC_LuCIn_5.UAct	;				
	emC_PPC[PPCNum].LuC[5].In.FAct	:=	emC_PPC_LuCIn_5.FAct	;				
	emC_PPC[PPCNum].LuC[5].In.PAct	:=	emC_PPC_LuCIn_5.PAct	;				
	emC_PPC[PPCNum].LuC[5].In.QAct	:=	emC_PPC_LuCIn_5.QAct	;				
	emC_PPC[PPCNum].LuC[5].In.TempAct	:=	emC_PPC_LuCIn_5.TempAct	;
							
						
					
END_PROGRAM

PROGRAM emC_PPC_R02_Sum
  VAR_EXTERNAL
    emC_PPC : emC_PPC_Array;
    PPCNum : INT;
    NbOfLuCPa : INT;
    NbOfBankPa : INT;
  END_VAR
  VAR
    L1_SPI_IN_1 : SPI_IN;
    L1_SPI_IN_2 : SPI_IN;
    L1_SPI_IN_3 : SPI_IN;
    L1_SPI_IN_4 : SPI_IN;
    L1_SPI_IN_5 : SPI_IN;
    L1_SPI_IN_6 : SPI_IN;
    L1_SPI_IN_7 : SPI_IN;
    L1_GCFaultSt_I : SPI;
    L1_NonCriticalAlarm_I : SPI;
    L1_CriticalAlarm_I : SPI;
    L1_Warning_I : SPI;
    L1_StoppingSt_I : SPI;
    L1_CtrlSystemReady_I : SPI;
    L1_BlackSys_I : SPI;
    L1_BatPNomMaxAct_I : MFI;
    L1_BatPNomMinAct_I : MFI;
    L1_SocPctAct_I : MFI;
    L1_UAct_I : MFI;
    L1_FAct_I : MFI;
    L1_PAct_I : MFI;
    L1_QAct_I : MFI;
    L1_TempAct_I : MFI;
    L1_MFI_IN_1 : MFI_IN;
    L1_MFI_IN_2 : MFI_IN;
    L1_MFI_IN_3 : MFI_IN;
    L1_MFI_IN_4 : MFI_IN;
    L1_MFI_IN_5 : MFI_IN;
    L1_MFI_IN_6 : MFI_IN;
    L1_MFI_IN_7 : MFI_IN;
    L1_MFI_IN_8 : MFI_IN;
    L2_SPI_IN_1 : SPI_IN;
    L2_SPI_IN_2 : SPI_IN;
    L2_SPI_IN_3 : SPI_IN;
    L2_SPI_IN_4 : SPI_IN;
    L2_SPI_IN_5 : SPI_IN;
    L2_SPI_IN_6 : SPI_IN;
    L2_SPI_IN_7 : SPI_IN;
    L2_GCFaultSt_I : SPI;
    L2_NonCriticalAlarm_I : SPI;
    L2_CriticalAlarm_I : SPI;
    L2_Warning_I : SPI;
    L2_StoppingSt_I : SPI;
    L2_CtrlSystemReady_I : SPI;
    L2_BlackSys_I : SPI;
    L2_BatPNomMaxAct_I : MFI;
    L2_BatPNomMinAct_I : MFI;
    L2_SocPctAct_I : MFI;
    L2_UAct_I : MFI;
    L2_FAct_I : MFI;
    L2_PAct_I : MFI;
    L2_QAct_I : MFI;
    L2_TempAct_I : MFI;
    L2_MFI_IN_1 : MFI_IN;
    L2_MFI_IN_2 : MFI_IN;
    L2_MFI_IN_3 : MFI_IN;
    L2_MFI_IN_4 : MFI_IN;
    L2_MFI_IN_5 : MFI_IN;
    L2_MFI_IN_6 : MFI_IN;
    L2_MFI_IN_7 : MFI_IN;
    L2_MFI_IN_8 : MFI_IN;
    L3_SPI_IN_1 : SPI_IN;
    L3_SPI_IN_2 : SPI_IN;
    L3_SPI_IN_3 : SPI_IN;
    L3_SPI_IN_4 : SPI_IN;
    L3_SPI_IN_5 : SPI_IN;
    L3_SPI_IN_6 : SPI_IN;
    L3_SPI_IN_7 : SPI_IN;
    L3_MFI_IN_1 : MFI_IN;
    L3_MFI_IN_2 : MFI_IN;
    L3_MFI_IN_3 : MFI_IN;
    L3_MFI_IN_4 : MFI_IN;
    L3_MFI_IN_5 : MFI_IN;
    L3_MFI_IN_6 : MFI_IN;
    L3_MFI_IN_7 : MFI_IN;
    L3_MFI_IN_8 : MFI_IN;
    L3_GCFaultSt_I : SPI;
    L3_NonCriticalAlarm_I : SPI;
    L3_CriticalAlarm_I : SPI;
    L3_Warning_I : SPI;
    L3_StoppingSt_I : SPI;
    L3_CtrlSystemReady_I : SPI;
    L3_BlackSys_I : SPI;
    L3_BatPNomMaxAct_I : MFI;
    L3_BatPNomMinAct_I : MFI;
    L3_SocPctAct_I : MFI;
    L3_UAct_I : MFI;
    L3_FAct_I : MFI;
    L3_PAct_I : MFI;
    L3_QAct_I : MFI;
    L3_TempAct_I : MFI;
    L4_SPI_IN_1 : SPI_IN;
    L4_SPI_IN_2 : SPI_IN;
    L4_SPI_IN_3 : SPI_IN;
    L4_SPI_IN_4 : SPI_IN;
    L4_SPI_IN_5 : SPI_IN;
    L4_SPI_IN_6 : SPI_IN;
    L4_SPI_IN_7 : SPI_IN;
    L4_MFI_IN_1 : MFI_IN;
    L4_MFI_IN_2 : MFI_IN;
    L4_MFI_IN_3 : MFI_IN;
    L4_MFI_IN_4 : MFI_IN;
    L4_MFI_IN_5 : MFI_IN;
    L4_MFI_IN_6 : MFI_IN;
    L4_MFI_IN_7 : MFI_IN;
    L4_MFI_IN_8 : MFI_IN;
    L4_GCFaultSt_I : SPI;
    L4_NonCriticalAlarm_I : SPI;
    L4_CriticalAlarm_I : SPI;
    L4_Warning_I : SPI;
    L4_StoppingSt_I : SPI;
    L4_CtrlSystemReady_I : SPI;
    L4_BlackSys_I : SPI;
    L4_BatPNomMaxAct_I : MFI;
    L4_BatPNomMinAct_I : MFI;
    L4_SocPctAct_I : MFI;
    L4_UAct_I : MFI;
    L4_FAct_I : MFI;
    L4_PAct_I : MFI;
    L4_QAct_I : MFI;
    L4_TempAct_I : MFI;
    L5_SPI_IN_1 : SPI_IN;
    L5_SPI_IN_2 : SPI_IN;
    L5_SPI_IN_3 : SPI_IN;
    L5_SPI_IN_4 : SPI_IN;
    L5_SPI_IN_5 : SPI_IN;
    L5_SPI_IN_6 : SPI_IN;
    L5_SPI_IN_7 : SPI_IN;
    L5_MFI_IN_1 : MFI_IN;
    L5_MFI_IN_2 : MFI_IN;
    L5_MFI_IN_3 : MFI_IN;
    L5_MFI_IN_4 : MFI_IN;
    L5_MFI_IN_5 : MFI_IN;
    L5_MFI_IN_6 : MFI_IN;
    L5_MFI_IN_7 : MFI_IN;
    L5_MFI_IN_8 : MFI_IN;
    L5_GCFaultSt_I : SPI;
    L5_NonCriticalAlarm_I : SPI;
    L5_CriticalAlarm_I : SPI;
    L5_Warning_I : SPI;
    L5_StoppingSt_I : SPI;
    L5_CtrlSystemReady_I : SPI;
    L5_BlackSys_I : SPI;
    L5_BatPNomMaxAct_I : MFI;
    L5_BatPNomMinAct_I : MFI;
    L5_SocPctAct_I : MFI;
    L5_UAct_I : MFI;
    L5_FAct_I : MFI;
    L5_PAct_I : MFI;
    L5_QAct_I : MFI;
    L5_TempAct_I : MFI;
    L6_SPI_IN_1 : SPI_IN;
    L6_SPI_IN_2 : SPI_IN;
    L6_SPI_IN_3 : SPI_IN;
    L6_SPI_IN_4 : SPI_IN;
    L6_SPI_IN_5 : SPI_IN;
    L6_SPI_IN_6 : SPI_IN;
    L6_SPI_IN_7 : SPI_IN;
    L6_MFI_IN_1 : MFI_IN;
    L6_MFI_IN_2 : MFI_IN;
    L6_MFI_IN_3 : MFI_IN;
    L6_MFI_IN_4 : MFI_IN;
    L6_MFI_IN_5 : MFI_IN;
    L6_MFI_IN_6 : MFI_IN;
    L6_MFI_IN_7 : MFI_IN;
    L6_MFI_IN_8 : MFI_IN;
    L6_GCFaultSt_I : SPI;
    L6_NonCriticalAlarm_I : SPI;
    L6_CriticalAlarm_I : SPI;
    L6_Warning_I : SPI;
    L6_StoppingSt_I : SPI;
    L6_CtrlSystemReady_I : SPI;
    L6_BlackSys_I : SPI;
    L6_BatPNomMaxAct_I : MFI;
    L6_BatPNomMinAct_I : MFI;
    L6_SocPctAct_I : MFI;
    L6_UAct_I : MFI;
    L6_FAct_I : MFI;
    L6_PAct_I : MFI;
    L6_QAct_I : MFI;
    L6_TempAct_I : MFI;
    L7_SPI_IN_1 : SPI_IN;
    L7_SPI_IN_2 : SPI_IN;
    L7_SPI_IN_3 : SPI_IN;
    L7_SPI_IN_4 : SPI_IN;
    L7_SPI_IN_5 : SPI_IN;
    L7_SPI_IN_6 : SPI_IN;
    L7_SPI_IN_7 : SPI_IN;
    L7_MFI_IN_1 : MFI_IN;
    L7_MFI_IN_2 : MFI_IN;
    L7_MFI_IN_3 : MFI_IN;
    L7_MFI_IN_4 : MFI_IN;
    L7_MFI_IN_5 : MFI_IN;
    L7_MFI_IN_6 : MFI_IN;
    L7_MFI_IN_7 : MFI_IN;
    L7_MFI_IN_8 : MFI_IN;
    L7_GCFaultSt_I : SPI;
    L7_NonCriticalAlarm_I : SPI;
    L7_CriticalAlarm_I : SPI;
    L7_Warning_I : SPI;
    L7_StoppingSt_I : SPI;
    L7_CtrlSystemReady_I : SPI;
    L7_BlackSys_I : SPI;
    L7_BatPNomMaxAct_I : MFI;
    L7_BatPNomMinAct_I : MFI;
    L7_SocPctAct_I : MFI;
    L7_UAct_I : MFI;
    L7_FAct_I : MFI;
    L7_PAct_I : MFI;
    L7_QAct_I : MFI;
    L7_TempAct_I : MFI;
    L8_SPI_IN_1 : SPI_IN;
    L8_SPI_IN_2 : SPI_IN;
    L8_SPI_IN_3 : SPI_IN;
    L8_SPI_IN_4 : SPI_IN;
    L8_SPI_IN_5 : SPI_IN;
    L8_SPI_IN_6 : SPI_IN;
    L8_SPI_IN_7 : SPI_IN;
    L8_MFI_IN_1 : MFI_IN;
    L8_MFI_IN_2 : MFI_IN;
    L8_MFI_IN_3 : MFI_IN;
    L8_MFI_IN_4 : MFI_IN;
    L8_MFI_IN_5 : MFI_IN;
    L8_MFI_IN_6 : MFI_IN;
    L8_MFI_IN_7 : MFI_IN;
    L8_MFI_IN_8 : MFI_IN;
    L8_GCFaultSt_I : SPI;
    L8_NonCriticalAlarm_I : SPI;
    L8_CriticalAlarm_I : SPI;
    L8_Warning_I : SPI;
    L8_StoppingSt_I : SPI;
    L8_CtrlSystemReady_I : SPI;
    L8_BlackSys_I : SPI;
    L8_BatPNomMaxAct_I : MFI;
    L8_BatPNomMinAct_I : MFI;
    L8_SocPctAct_I : MFI;
    L8_UAct_I : MFI;
    L8_FAct_I : MFI;
    L8_PAct_I : MFI;
    L8_QAct_I : MFI;
    L8_TempAct_I : MFI;
  END_VAR

						
							emC_PPC[PPCNum].Summary.ComFaultCnt	:=	0	;		
emC_PPC[PPCNum].Summary.OnlineCnt	:=	0	;
emC_PPC[PPCNum].Summary.AvgTempAct	:=	REAL#0.0	;
emC_PPC[PPCNum].Summary.TotBatPNomMaxAct	:=	REAL#0.0	;
emC_PPC[PPCNum].Summary.TotBatPNomMinAct	:=	REAL#0.0	;
emC_PPC[PPCNum].Summary.AvgSocPct	:=	REAL#0.0	;
emC_PPC[PPCNum].Summary.AvgUAct	:=	REAL#0.0	;
emC_PPC[PPCNum].Summary.AvgFAct	:=	REAL#0.0	;
emC_PPC[PPCNum].Summary.TotPAct	:=	REAL#0.0	;
emC_PPC[PPCNum].Summary.TotQAct	:=	REAL#0.0	;
	
								
